KUKA KRL program: MyProgram_207().src

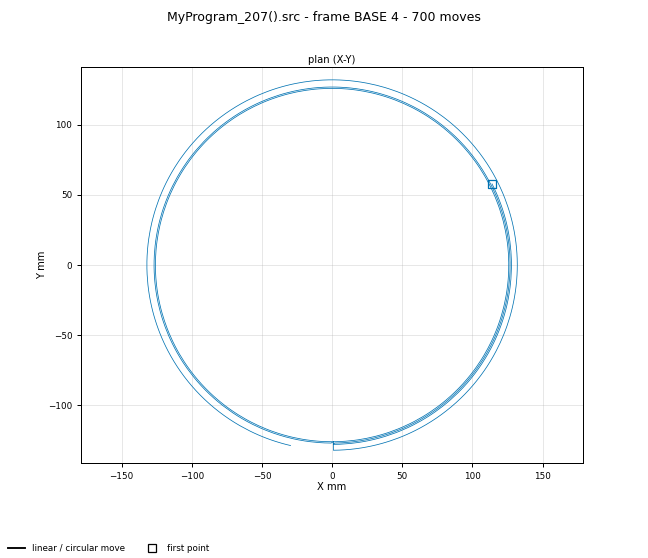
[picture p0: tool path of MyProgram_207().src in frame BASE 4, 700 of 700 moves have a stored position in this frame; points joined in program order, loops and branches not executed]
&ACCESS RVP
&REL 1
&PARAM TEMPLATE = C:\KRC\Roboter\Template\vorgabe
&PARAM EDITMASK = *
DEF MyProgram_207()
; ---- Setting reference (Base) ----
$BASE = BASE_DATA[4]

; --------------------------
; ---- Setting tool (TCP) ----
$TOOL = TOOL_DATA[3]
; --------------------------

$VEL.CP = VEL_APROX_PRINT
Startdeposition()
$VEL.CP = VEL_PRINT
LIN {X 113.9703,Y 57.8056,Z 147,A 23.526,B 22.3561,C -1.1422,E1 22.5268,E2 423.6264} C_DIS
LIN {X 115.5731,Y 54.5336,Z 147,A 21.9006,B 22.3563,C -1.138,E1 22.5287,E2 425.2529} C_DIS
LIN {X 117.0607,Y 51.2625,Z 147,A 19.7387,B 22.3577,C -1.1077,E1 22.5312,E2 427.4806} C_DIS
LIN {X 118.7833,Y 47.134,Z 147,A 18.1732,B 22.357,C -1.1224,E1 22.5328,E2 428.9979} C_DIS
LIN {X 120.2237,Y 43.3241,Z 147,A 16.48,B 22.357,C -1.1233,E1 22.5344,E2 430.6782} C_DIS
LIN {X 121.3863,Y 39.9534,Z 147,A 14.784,B 22.3574,C -1.1139,E1 22.536,E2 432.3878} C_DIS
LIN {X 122.6165,Y 35.9988,Z 147,A 13.0614,B 22.3574,C -1.1146,E1 22.5374,E2 434.0973} C_DIS
LIN {X 123.4639,Y 32.9755,Z 147,A 11.6527,B 22.3576,C -1.1103,E1 22.5384,E2 435.5083} C_DIS
LIN {X 124.3219,Y 29.5794,Z 147,A 9.9835,B 22.358,C -1.1008,E1 22.5395,E2 437.1913} C_DIS
LIN {X 125.2135,Y 25.5406,Z 147,A 8.2593,B 22.358,C -1.1012,E1 22.5405,E2 438.9031} C_DIS
LIN {X 125.8843,Y 22.0036,Z 147,A 6.6854,B 22.3582,C -1.0981,E1 22.5413,E2 440.4749} C_DIS
LIN {X 126.6501,Y 17.0512,Z 147,A 4.3479,B 22.3587,C -1.0867,E1 22.5423,E2 442.8265} C_DIS
LIN {X 127.4072,Y 9.93,Z 147,A 1.3243,B 22.3587,C -1.0853,E1 22.5431,E2 445.8334} C_DIS
LIN {X 127.7553,Y 3.0983,Z 147,A -1.7197,B 22.3592,C -1.0766,E1 22.5435,E2 448.8798} C_DIS
LIN {X 127.7807,Y -1.7513,Z 147,A -3.7775,B 22.3592,C -1.0751,E1 22.5435,E2 450.9276} C_DIS
LIN {X 127.4011,Y -10.0131,Z 147,A -7.5963,B 22.36,C -1.0579,E1 22.543,E2 454.7657} C_DIS
LIN {X 126.813,Y -15.8021,Z 147,A -10.1858,B 22.3603,C -1.0504,E1 22.5422,E2 457.3574} C_DIS
LIN {X 126.3725,Y -19.0018,Z 147,A -12.4156,B 22.3622,C -1.0089,E1 22.5412,E2 459.6807} C_DIS
LIN {X 125.461,Y -24.2979,Z 147,A -14.1841,B 22.3612,C -1.0313,E1 22.5404,E2 461.3788} C_DIS
LIN {X 124.5922,Y -28.417,Z 147,A -15.9529,B 22.3612,C -1.031,E1 22.5393,E2 463.137} C_DIS
LIN {X 123.828,Y -31.5812,Z 147,A -17.4094,B 22.3614,C -1.0265,E1 22.5383,E2 464.5956} C_DIS
LIN {X 122.7533,Y -35.5317,Z 147,A -19.2625,B 22.3617,C -1.0199,E1 22.5369,E2 466.454} C_DIS
LIN {X 121.6682,Y -39.0845,Z 147,A -20.8504,B 22.3617,C -1.0184,E1 22.5356,E2 468.0357} C_DIS
LIN {X 120.617,Y -42.2183,Z 147,A -22.4583,B 22.3622,C -1.0078,E1 22.5341,E2 469.6609} C_DIS
LIN {X 119.0143,Y -46.5442,Z 147,A -24.3866,B 22.3622,C -1.0081,E1 22.5322,E2 471.5763} C_DIS
LIN {X 117.6766,Y -49.8329,Z 147,A -25.9364,B 22.3623,C -1.0052,E1 22.5306,E2 473.124} C_DIS
LIN {X 116.3291,Y -52.904,Z 147,A -27.4435,B 22.3625,C -1.0005,E1 22.5289,E2 474.6342} C_DIS
LIN {X 115.0029,Y -55.7271,Z 147,A -29.3445,B 22.3637,C -0.9726,E1 22.5265,E2 476.5963} C_DIS
LIN {X 113.1768,Y -59.3438,Z 147,A -30.5723,B 22.3627,C -0.995,E1 22.525,E2 477.7583} C_DIS
LIN {X 111.2715,Y -62.8481,Z 147,A -32.8273,B 22.3639,C -0.9678,E1 22.5219,E2 480.071} C_DIS
LIN {X 109.42,Y -66.0186,Z 147,A -34.0958,B 22.3633,C -0.9809,E1 22.5201,E2 481.2982} C_DIS
LIN {X 106.5876,Y -70.5006,Z 147,A -36.4479,B 22.3636,C -0.9753,E1 22.5165,E2 483.6513} C_DIS
LIN {X 104.3333,Y -73.7954,Z 147,A -38.2742,B 22.3638,C -0.9687,E1 22.5136,E2 485.4848} C_DIS
LIN {X 101.8263,Y -77.2183,Z 147,A -40.7015,B 22.365,C -0.939,E1 22.5094,E2 487.9765} C_DIS
LIN {X 98.9094,Y -80.9204,Z 147,A -42.2776,B 22.3643,C -0.9585,E1 22.5068,E2 489.4933} C_DIS
LIN {X 96.1295,Y -84.2042,Z 147,A -44.5875,B 22.3652,C -0.9358,E1 22.5025,E2 491.8508} C_DIS
LIN {X 93.4028,Y -87.2188,Z 147,A -46.6124,B 22.3657,C -0.9219,E1 22.4985,E2 493.9021} C_DIS
LIN {X 89.8071,Y -90.9174,Z 147,A -48.0288,B 22.3643,C -0.958,E1 22.496,E2 495.2173} C_DIS
LIN {X 84.1748,Y -96.1551,Z 147,A -52.1641,B 22.3659,C -0.918,E1 22.4873,E2 499.4382} C_DIS
LIN {X 80.94,Y -98.8933,Z 147,A -53.3106,B 22.3646,C -0.9488,E1 22.485,E2 500.4992} C_DIS
LIN {X 78.6247,Y -100.7446,Z 147,A -54.9716,B 22.3654,C -0.9305,E1 22.4812,E2 502.2012} C_DIS
LIN {X 73.4716,Y -104.5617,Z 147,A -57.9316,B 22.3658,C -0.9207,E1 22.4745,E2 505.1751} C_DIS
LIN {X 70.6355,Y -106.4986,Z 147,A -59.2877,B 22.3655,C -0.9261,E1 22.4714,E2 506.5117} C_DIS
LIN {X 67.4689,Y -108.5317,Z 147,A -61.575,B 22.3667,C -0.8954,E1 22.4658,E2 508.8713} C_DIS
LIN {X 63.2901,Y -111.0204,Z 147,A -63.0555,B 22.3656,C -0.9236,E1 22.4625,E2 510.2728} C_DIS
LIN {X 60.2184,Y -112.7158,Z 147,A -64.7771,B 22.366,C -0.914,E1 22.4582,E2 512.0138} C_DIS
LIN {X 57.6094,Y -114.0702,Z 147,A -66.0145,B 22.366,C -0.9156,E1 22.4551,E2 513.2433} C_DIS
LIN {X 53.8834,Y -115.8764,Z 147,A -67.9484,B 22.3662,C -0.9091,E1 22.4502,E2 515.1884} C_DIS
LIN {X 47.9039,Y -118.4733,Z 147,A -70.4708,B 22.3657,C -0.9232,E1 22.4439,E2 517.667} C_DIS
LIN {X 45.3901,Y -119.4605,Z 147,A -72.0569,B 22.3664,C -0.9044,E1 22.4396,E2 519.2987} C_DIS
LIN {X 37.9509,Y -122.0278,Z 147,A -75.5995,B 22.3666,C -0.8994,E1 22.4302,E2 522.8465} C_DIS
LIN {X 34.2312,Y -123.1219,Z 147,A -77.2411,B 22.3665,C -0.9019,E1 22.4258,E2 524.4784} C_DIS
LIN {X 30.1666,Y -124.1804,Z 147,A -79.1021,B 22.3665,C -0.901,E1 22.4208,E2 526.3384} C_DIS
LIN {X 26.8694,Y -124.9351,Z 147,A -80.6062,B 22.3665,C -0.9002,E1 22.4167,E2 527.8424} C_DIS
LIN {X 23.5519,Y -125.6036,Z 147,A -82.0308,B 22.3665,C -0.9032,E1 22.4128,E2 529.2574} C_DIS
LIN {X 19.255,Y -126.3333,Z 147,A -84.2028,B 22.3669,C -0.8919,E1 22.4068,E2 531.4563} C_DIS
LIN {X 12.928,Y -127.1384,Z 147,A -86.9402,B 22.3667,C -0.8957,E1 22.3992,E2 534.1816} C_DIS
LIN {X 5.1547,Y -127.6882,Z 147,A -90.1483,B 22.3663,C -0.907,E1 22.3904,E2 537.3584} C_DIS
LIN {X 0.9063,Y -127.7615,Z 147,A -91.5691,B 22.3655,C -0.9285,E1 22.3866,E2 538.7223} C_DIS
Enddeposition()
LIN {X 0.9063,Y -127.7615,Z 147,A -91.5691,B 22.3655,C -0.9285,E1 22.3866,E2 538.7223} C_DIS
Startdeposition()
$VEL.CP = VEL_PRINT
LIN {X 1.8845,Y -126.8238,Z 147,A -90.6214,B 21.3631,C -0.7912,E1 21.3818,E2 538.0225} C_DIS
LIN {X 7.2855,Y -126.6292,Z 147,A -88.1843,B 21.3631,C -0.7918,E1 21.3886,E2 535.5846} C_DIS
LIN {X 12.6919,Y -126.2022,Z 147,A -85.9631,B 21.3634,C -0.7832,E1 21.3947,E2 533.3886} C_DIS
LIN {X 16.8635,Y -125.712,Z 147,A -83.7531,B 21.3628,C -0.7978,E1 21.4009,E2 531.1405} C_DIS
LIN {X 20.3755,Y -125.1911,Z 147,A -82.5082,B 21.3633,C -0.7834,E1 21.4042,E2 529.9366} C_DIS
LIN {X 23.4283,Y -124.6555,Z 147,A -81.3063,B 21.3636,C -0.7759,E1 21.4075,E2 528.7568} C_DIS
LIN {X 26.5889,Y -124.0192,Z 147,A -79.7344,B 21.3634,C -0.7822,E1 21.4118,E2 527.1701} C_DIS
LIN {X 29.316,Y -123.4036,Z 147,A -78.4117,B 21.3633,C -0.7859,E1 21.4154,E2 525.8395} C_DIS
LIN {X 32.5994,Y -122.5764,Z 147,A -76.8881,B 21.3633,C -0.7872,E1 21.4195,E2 524.3152} C_DIS
LIN {X 35.485,Y -121.7724,Z 147,A -75.6426,B 21.3633,C -0.7839,E1 21.4229,E2 523.081} C_DIS
LIN {X 38.1101,Y -120.9775,Z 147,A -73.9866,B 21.3626,C -0.8036,E1 21.4274,E2 521.3749} C_DIS
LIN {X 41.1624,Y -119.9729,Z 147,A -72.9028,B 21.3631,C -0.7892,E1 21.4302,E2 520.3329} C_DIS
LIN {X 44.4417,Y -118.7965,Z 147,A -71.4954,B 21.3633,C -0.784,E1 21.4338,E2 518.9434} C_DIS
LIN {X 47.2457,Y -117.7095,Z 147,A -70.1052,B 21.3633,C -0.7872,E1 21.4374,E2 517.548} C_DIS
LIN {X 50.7884,Y -116.2258,Z 147,A -67.8469,B 21.3623,C -0.8127,E1 21.4434,E2 515.2264} C_DIS
LIN {X 54.006,Y -114.7673,Z 147,A -66.4973,B 21.3626,C -0.8042,E1 21.4467,E2 513.9041} C_DIS
LIN {X 57.2234,Y -113.1956,Z 147,A -65.1958,B 21.363,C -0.7929,E1 21.4499,E2 512.6378} C_DIS
LIN {X 61.1503,Y -111.1255,Z 147,A -62.9133,B 21.3625,C -0.8085,E1 21.4556,E2 510.3204} C_DIS
LIN {X 66.7546,Y -107.852,Z 147,A -59.9734,B 21.3623,C -0.8141,E1 21.4627,E2 507.3759} C_DIS
LIN {X 70.0235,Y -105.7589,Z 147,A -58.2251,B 21.3621,C -0.8172,E1 21.4668,E2 505.626} C_DIS
LIN {X 72.9782,Y -103.7416,Z 147,A -56.6366,B 21.3621,C -0.8192,E1 21.4704,E2 504.0386} C_DIS
LIN {X 76.3709,Y -101.2699,Z 147,A -54.7572,B 21.362,C -0.8223,E1 21.4746,E2 502.1586} C_DIS
LIN {X 79.7116,Y -98.662,Z 147,A -52.906,B 21.362,C -0.8236,E1 21.4787,E2 500.3121} C_DIS
LIN {X 82.6549,Y -96.2098,Z 147,A -51.1096,B 21.3617,C -0.8303,E1 21.4825,E2 498.5056} C_DIS
LIN {X 86.242,Y -93.0081,Z 147,A -48.9386,B 21.3615,C -0.8353,E1 21.487,E2 496.3316} C_DIS
LIN {X 89.5793,Y -89.7983,Z 147,A -46.939,B 21.3615,C -0.8361,E1 21.491,E2 494.3397} C_DIS
LIN {X 93.0775,Y -86.1675,Z 147,A -44.5379,B 21.361,C -0.8472,E1 21.4956,E2 491.9207} C_DIS
LIN {X 96.2028,Y -82.6629,Z 147,A -42.5135,B 21.361,C -0.8482,E1 21.4993,E2 489.9044} C_DIS
LIN {X 98.9918,Y -79.3025,Z 147,A -40.8259,B 21.3613,C -0.8404,E1 21.5023,E2 488.2473} C_DIS
LIN {X 101.0125,Y -76.712,Z 147,A -39.0644,B 21.3607,C -0.8569,E1 21.5053,E2 486.4509} C_DIS
LIN {X 103.1861,Y -73.7614,Z 147,A -37.4465,B 21.3606,C -0.8596,E1 21.508,E2 484.8348} C_DIS
LIN {X 105.6815,Y -70.1403,Z 147,A -35.7291,B 21.3608,C -0.8529,E1 21.5106,E2 483.1459} C_DIS
LIN {X 107.4069,Y -67.4682,Z 147,A -34.0362,B 21.3602,C -0.8685,E1 21.5132,E2 481.4205} C_DIS
LIN {X 109.394,Y -64.1956,Z 147,A -32.5953,B 21.3605,C -0.8603,E1 21.5152,E2 480.0108} C_DIS
LIN {X 110.9698,Y -61.4314,Z 147,A -30.9238,B 21.36,C -0.875,E1 21.5176,E2 478.3094} C_DIS
LIN {X 113.1495,Y -57.3139,Z 147,A -28.8604,B 21.3598,C -0.8793,E1 21.5202,E2 476.2473} C_DIS
LIN {X 115.0671,Y -53.3593,Z 147,A -27.0683,B 21.3599,C -0.8764,E1 21.5224,E2 474.4747} C_DIS
LIN {X 116.2361,Y -50.7645,Z 147,A -25.578,B 21.3594,C -0.8895,E1 21.5241,E2 472.9583} C_DIS
LIN {X 117.5184,Y -47.7198,Z 147,A -24.3391,B 21.3597,C -0.8825,E1 21.5254,E2 471.7466} C_DIS
LIN {X 118.7816,Y -44.4815,Z 147,A -22.5752,B 21.3591,C -0.8961,E1 21.5271,E2 469.9573} C_DIS
LIN {X 120.1599,Y -40.6152,Z 147,A -20.6624,B 21.3588,C -0.9044,E1 21.5289,E2 468.0346} C_DIS
LIN {X 121.2727,Y -37.1565,Z 147,A -19.1074,B 21.3588,C -0.9056,E1 21.5302,E2 466.487} C_DIS
LIN {X 122.4349,Y -33.1301,Z 147,A -17.3559,B 21.3588,C -0.905,E1 21.5315,E2 464.749} C_DIS
LIN {X 123.1502,Y -30.367,Z 147,A -16.0335,B 21.3585,C -0.9105,E1 21.5324,E2 463.4205} C_DIS
LIN {X 123.8046,Y -27.5787,Z 147,A -14.5825,B 21.3581,C -0.9218,E1 21.5333,E2 461.9489} C_DIS
LIN {X 124.5256,Y -24.1076,Z 147,A -13.2442,B 21.3584,C -0.9148,E1 21.5341,E2 460.6388} C_DIS
LIN {X 125.241,Y -20.0715,Z 147,A -11.1576,B 21.3577,C -0.9314,E1 21.535,E2 458.5217} C_DIS
LIN {X 125.7775,Y -16.3637,Z 147,A -9.505,B 21.3575,C -0.935,E1 21.5357,E2 456.8709} C_DIS
LIN {X 126.3404,Y -11.2331,Z 147,A -7.2906,B 21.3575,C -0.937,E1 21.5363,E2 454.6665} C_DIS
LIN {X 126.5367,Y -8.7446,Z 147,A -5.9494,B 21.3569,C -0.9504,E1 21.5366,E2 453.2984} C_DIS
LIN {X 126.7698,Y -4.2032,Z 147,A -4.0657,B 21.3569,C -0.9491,E1 21.5368,E2 451.4315} C_DIS
LIN {X 126.8383,Y -0.4449,Z 147,A -2.4296,B 21.3569,C -0.9517,E1 21.5368,E2 449.7999} C_DIS
LIN {X 126.8228,Y 1.9441,Z 147,A -1.1678,B 21.3563,C -0.9635,E1 21.5368,E2 448.5149} C_DIS
LIN {X 126.6093,Y 7.6081,Z 147,A 1.183,B 21.3563,C -0.962,E1 21.5365,E2 446.1847} C_DIS
LIN {X 126.3642,Y 10.9505,Z 147,A 2.5647,B 21.3564,C -0.9608,E1 21.5362,E2 444.8161} C_DIS
LIN {X 125.9929,Y 14.6184,Z 147,A 4.1603,B 21.3564,C -0.9628,E1 21.5357,E2 443.2262} C_DIS
LIN {X 125.5699,Y 17.887,Z 147,A 5.8153,B 21.3558,C -0.975,E1 21.5351,E2 441.5495} C_DIS
LIN {X 124.9578,Y 21.7628,Z 147,A 7.5122,B 21.3558,C -0.9771,E1 21.5343,E2 439.8588} C_DIS
LIN {X 124.317,Y 25.1597,Z 147,A 9.1797,B 21.3553,C -0.9867,E1 21.5334,E2 438.1766} C_DIS
LIN {X 123.3874,Y 29.3829,Z 147,A 11.0808,B 21.3552,C -0.9903,E1 21.5322,E2 436.2788} C_DIS
LIN {X 122.4672,Y 33.0088,Z 147,A 12.7925,B 21.3549,C -0.9964,E1 21.531,E2 434.5622} C_DIS
LIN {X 121.3235,Y 36.9907,Z 147,A 14.5965,B 21.3548,C -0.999,E1 21.5296,E2 432.7635} C_DIS
LIN {X 120.3315,Y 40.1,Z 147,A 16.0349,B 21.3546,C -1.0018,E1 21.5283,E2 431.3273} C_DIS
LIN {X 119.4191,Y 42.7414,Z 147,A 17.5096,B 21.354,C -1.0151,E1 21.5269,E2 429.8261} C_DIS
LIN {X 117.6039,Y 47.5077,Z 147,A 19.9226,B 21.3535,C -1.0267,E1 21.5244,E2 427.3974} C_DIS
LIN {X 116.3271,Y 50.5539,Z 147,A 21.1514,B 21.3539,C -1.019,E1 21.5231,E2 426.1974} C_DIS
LIN {X 114.8228,Y 53.8878,Z 147,A 22.869,B 21.3535,C -1.0266,E1 21.5211,E2 424.4703} C_DIS
LIN {X 113.0711,Y 57.4679,Z 147,A 24.4916,B 21.3537,C -1.0236,E1 21.5191,E2 422.8661} C_DIS
LIN {X 111.6437,Y 60.1984,Z 147,A 25.8184,B 21.3537,C -1.0244,E1 21.5174,E2 421.5454} C_DIS
LIN {X 109.4873,Y 64.0369,Z 147,A 28.4643,B 21.352,C -1.0593,E1 21.5136,E2 418.8205} C_DIS
LIN {X 107.0602,Y 68.0174,Z 147,A 29.975,B 21.353,C -1.038,E1 21.5114,E2 417.3771} C_DIS
LIN {X 104.8819,Y 71.3301,Z 147,A 31.8198,B 21.3527,C -1.045,E1 21.5085,E2 415.5242} C_DIS
LIN {X 102.4325,Y 74.8053,Z 147,A 33.7868,B 21.3524,C -1.0518,E1 21.5053,E2 413.5499} C_DIS
LIN {X 99.6595,Y 78.461,Z 147,A 35.7435,B 21.3524,C -1.0516,E1 21.502,E2 411.6046} C_DIS
LIN {X 97.1625,Y 81.5326,Z 147,A 37.5801,B 21.3521,C -1.058,E1 21.4987,E2 409.7608} C_DIS
LIN {X 94.2164,Y 84.9209,Z 147,A 39.6131,B 21.3518,C -1.0628,E1 21.495,E2 407.7256} C_DIS
LIN {X 91.0186,Y 88.3389,Z 147,A 41.6737,B 21.3518,C -1.065,E1 21.491,E2 405.6694} C_DIS
LIN {X 87.95,Y 91.3951,Z 147,A 43.5616,B 21.3517,C -1.0661,E1 21.4872,E2 403.788} C_DIS
LIN {X 84.9836,Y 94.1595,Z 147,A 45.4795,B 21.3513,C -1.0736,E1 21.4833,E2 401.8588} C_DIS
LIN {X 81.8299,Y 96.9131,Z 147,A 47.3466,B 21.3512,C -1.0762,E1 21.4793,E2 399.9933} C_DIS
LIN {X 78.6628,Y 99.5009,Z 147,A 49.2351,B 21.3509,C -1.0815,E1 21.4752,E2 398.0989} C_DIS
LIN {X 75.0876,Y 102.2251,Z 147,A 51.2071,B 21.3509,C -1.0825,E1 21.4708,E2 396.1326} C_DIS
LIN {X 71.4256,Y 104.8173,Z 147,A 53.2675,B 21.3507,C -1.0874,E1 21.4661,E2 394.0672} C_DIS
LIN {X 67.7015,Y 107.2597,Z 147,A 55.0921,B 21.3509,C -1.0824,E1 21.4618,E2 392.2634} C_DIS
LIN {X 65.6014,Y 108.5568,Z 147,A 56.336,B 21.3505,C -1.0897,E1 21.4588,E2 391.0042} C_DIS
LIN {X 61.8107,Y 110.7597,Z 147,A 58.372,B 21.3503,C -1.0949,E1 21.4539,E2 388.9611} C_DIS
LIN {X 57.7877,Y 112.9083,Z 147,A 60.295,B 21.3504,C -1.0917,E1 21.4491,E2 387.0531} C_DIS
LIN {X 55.0999,Y 114.2447,Z 147,A 61.4922,B 21.3507,C -1.0866,E1 21.4462,E2 385.8739} C_DIS
LIN {X 52.5219,Y 115.4544,Z 147,A 63.0451,B 21.3501,C -1.0995,E1 21.4422,E2 384.2902} C_DIS
LIN {X 49.2412,Y 116.8893,Z 147,A 64.3472,B 21.3506,C -1.0878,E1 21.4389,E2 383.0239} C_DIS
LIN {X 46.1275,Y 118.1522,Z 147,A 65.891,B 21.3506,C -1.0905,E1 21.4349,E2 381.477} C_DIS
LIN {X 43.0582,Y 119.3049,Z 147,A 67.5406,B 21.3501,C -1.0991,E1 21.4305,E2 379.8079} C_DIS
LIN {X 39.4316,Y 120.5538,Z 147,A 69.7425,B 21.349,C -1.1206,E1 21.4246,E2 377.5521} C_DIS
LIN {X 35.589,Y 121.742,Z 147,A 71.0332,B 21.3501,C -1.0995,E1 21.4213,E2 376.3219} C_DIS
LIN {X 32.4444,Y 122.6177,Z 147,A 72.512,B 21.3501,C -1.1007,E1 21.4173,E2 374.8427} C_DIS
LIN {X 28.663,Y 123.557,Z 147,A 74.3242,B 21.3498,C -1.1039,E1 21.4123,E2 373.0248} C_DIS
LIN {X 25.4524,Y 124.2575,Z 147,A 75.8106,B 21.3498,C -1.1048,E1 21.4083,E2 371.5383} C_DIS
LIN {X 21.3949,Y 125.021,Z 147,A 77.6898,B 21.3498,C -1.1061,E1 21.4031,E2 369.6579} C_DIS
LIN {X 17.278,Y 125.6569,Z 147,A 79.6656,B 21.3495,C -1.1106,E1 21.3976,E2 367.6719} C_DIS
LIN {X 13.0799,Y 126.1622,Z 147,A 81.5158,B 21.3496,C -1.1085,E1 21.3925,E2 365.8291} C_DIS
LIN {X 9.368,Y 126.4912,Z 147,A 83.096,B 21.3498,C -1.1043,E1 21.3881,E2 364.2613} C_DIS
LIN {X 5.6663,Y 126.7127,Z 147,A 84.7258,B 21.3499,C -1.1024,E1 21.3836,E2 362.6374} C_DIS
LIN {X 2.5413,Y 126.8129,Z 147,A 86.3568,B 21.3495,C -1.1114,E1 21.379,E2 360.9821} C_DIS
LIN {X -1.518,Y 126.8299,Z 147,A 88.1668,B 21.3495,C -1.1101,E1 21.3739,E2 359.1757} C_DIS
LIN {X -5.6527,Y 126.7134,Z 147,A 90.1181,B 21.3494,C -1.113,E1 21.3685,E2 357.216} C_DIS
LIN {X -9.8605,Y 126.4552,Z 147,A 91.7492,B 21.35,C -1.101,E1 21.364,E2 355.6172} C_DIS
LIN {X -13.1058,Y 126.1594,Z 147,A 93.1324,B 21.3502,C -1.0967,E1 21.3602,E2 354.245} C_DIS
LIN {X -16.2644,Y 125.7905,Z 147,A 94.6679,B 21.35,C -1.1,E1 21.3559,E2 352.6992} C_DIS
LIN {X -20.7603,Y 125.1269,Z 147,A 96.4994,B 21.3505,C -1.0896,E1 21.3509,E2 350.8944} C_DIS
LIN {X -24.6616,Y 124.4184,Z 147,A 98.6423,B 21.3499,C -1.1026,E1 21.345,E2 348.713} C_DIS
LIN {X -27.7201,Y 123.7723,Z 147,A 100.1,B 21.3499,C -1.1033,E1 21.341,E2 347.2513} C_DIS
LIN {X -31.4319,Y 122.8812,Z 147,A 101.6902,B 21.3502,C -1.0962,E1 21.3367,E2 345.6778} C_DIS
LIN {X -35.0421,Y 121.9021,Z 147,A 103.4843,B 21.3501,C -1.0988,E1 21.3319,E2 343.8734} C_DIS
LIN {X -38.0352,Y 121.0014,Z 147,A 104.9052,B 21.3501,C -1.0976,E1 21.3281,E2 342.4528} C_DIS
LIN {X -41.575,Y 119.8298,Z 147,A 106.3171,B 21.3508,C -1.0846,E1 21.3244,E2 341.0733} C_DIS
LIN {X -44.3623,Y 118.8262,Z 147,A 107.8645,B 21.3505,C -1.0914,E1 21.3203,E2 339.5037} C_DIS
LIN {X -47.4629,Y 117.622,Z 147,A 109.3844,B 21.3505,C -1.0901,E1 21.3163,E2 337.9834} C_DIS
LIN {X -50.7011,Y 116.2635,Z 147,A 111.0935,B 21.3504,C -1.0928,E1 21.3119,E2 336.262} C_DIS
LIN {X -53.9719,Y 114.7836,Z 147,A 113.0422,B 21.3499,C -1.1035,E1 21.3069,E2 334.278} C_DIS
LIN {X -57.3652,Y 113.1234,Z 147,A 114.0368,B 21.3514,C -1.0724,E1 21.3047,E2 333.3661} C_DIS
LIN {X -61.889,Y 110.7155,Z 147,A 117.2537,B 21.3498,C -1.1046,E1 21.2965,E2 330.0496} C_DIS
LIN {X -66.0326,Y 108.2956,Z 147,A 118.9326,B 21.351,C -1.0811,E1 21.2926,E2 328.4292} C_DIS
LIN {X -69.6127,Y 106.0293,Z 147,A 120.8065,B 21.3512,C -1.076,E1 21.2883,E2 326.5623} C_DIS
LIN {X -73.3244,Y 103.4975,Z 147,A 122.7813,B 21.3515,C -1.0699,E1 21.2837,E2 324.5963} C_DIS
LIN {X -75.9784,Y 101.5652,Z 147,A 124.6517,B 21.3509,C -1.0822,E1 21.2795,E2 322.6838} C_DIS
LIN {X -78.8523,Y 99.3502,Z 147,A 125.9504,B 21.3517,C -1.0653,E1 21.2767,E2 321.4262} C_DIS
LIN {X -81.8169,Y 96.924,Z 147,A 127.5355,B 21.3522,C -1.0558,E1 21.2733,E2 319.8599} C_DIS
LIN {X -84.4057,Y 94.6778,Z 147,A 128.977,B 21.3525,C -1.0482,E1 21.2703,E2 318.4327} C_DIS
LIN {X -88.8116,Y 90.5573,Z 147,A 132.0462,B 21.3522,C -1.0554,E1 21.2641,E2 315.3286} C_DIS
LIN {X -91.657,Y 87.6762,Z 147,A 133.9648,B 21.3522,C -1.0545,E1 21.2603,E2 313.4025} C_DIS
LIN {X -97.3657,Y 81.2904,Z 147,A 137.7565,B 21.3528,C -1.0418,E1 21.2534,E2 309.6257} C_DIS
LIN {X -99.1912,Y 79.0521,Z 147,A 139.0671,B 21.353,C -1.0387,E1 21.2511,E2 308.3165} C_DIS
LIN {X -101.675,Y 75.8309,Z 147,A 140.8901,B 21.3532,C -1.0333,E1 21.248,E2 306.4979} C_DIS
LIN {X -103.4114,Y 73.4464,Z 147,A 142.3209,B 21.3532,C -1.0335,E1 21.2457,E2 305.0581} C_DIS
LIN {X -106.0078,Y 69.6454,Z 147,A 144.2176,B 21.3538,C -1.0208,E1 21.2427,E2 303.1854} C_DIS
LIN {X -108.5512,Y 65.6106,Z 147,A 146.4238,B 21.354,C -1.0168,E1 21.2395,E2 300.9768} C_DIS
LIN {X -110.3503,Y 62.5385,Z 147,A 148.1244,B 21.354,C -1.0158,E1 21.2371,E2 299.2684} C_DIS
LIN {X -112.2046,Y 59.1423,Z 147,A 149.723,B 21.3545,C -1.005,E1 21.235,E2 297.6895} C_DIS
LIN {X -113.5464,Y 56.525,Z 147,A 151.0007,B 21.3548,C -0.9992,E1 21.2334,E2 296.4197} C_DIS
LIN {X -115.2278,Y 53.0118,Z 147,A 153.0207,B 21.3545,C -1.0041,E1 21.231,E2 294.373} C_DIS
LIN {X -117.0658,Y 48.8187,Z 147,A 154.9862,B 21.355,C -0.9939,E1 21.2288,E2 292.4226} C_DIS
LIN {X -118.5773,Y 45.0267,Z 147,A 157.1165,B 21.3548,C -0.9994,E1 21.2267,E2 290.2629} C_DIS
LIN {X -120.1187,Y 40.739,Z 147,A 159.0352,B 21.3553,C -0.9877,E1 21.2249,E2 288.3636} C_DIS
LIN {X -121.198,Y 37.4006,Z 147,A 160.5298,B 21.3556,C -0.9794,E1 21.2237,E2 286.8818} C_DIS
LIN {X -122.871,Y 31.4722,Z 147,A 163.3581,B 21.3559,C -0.9725,E1 21.2216,E2 284.0529} C_DIS
LIN {X -123.6444,Y 28.2802,Z 147,A 164.7918,B 21.3562,C -0.9659,E1 21.2207,E2 282.6274} C_DIS
LIN {X -124.325,Y 25.1205,Z 147,A 166.4099,B 21.3562,C -0.9674,E1 21.2197,E2 280.9938} C_DIS
LIN {X -125.118,Y 20.8135,Z 147,A 168.3115,B 21.3566,C -0.9582,E1 21.2188,E2 279.1042} C_DIS
LIN {X -125.6629,Y 17.236,Z 147,A 170.0014,B 21.3566,C -0.9551,E1 21.2181,E2 277.4107} C_DIS
LIN {X -126.1089,Y 13.5752,Z 147,A 171.648,B 21.3569,C -0.9491,E1 21.2176,E2 275.769} C_DIS
LIN {X -126.4759,Y 9.5777,Z 147,A 173.3626,B 21.3573,C -0.9396,E1 21.2172,E2 274.0685} C_DIS
LIN {X -126.6451,Y 7.0145,Z 147,A 174.7931,B 21.3571,C -0.9463,E1 21.217,E2 272.6092} C_DIS
LIN {X -126.804,Y 2.9711,Z 147,A 176.5928,B 21.3573,C -0.9394,E1 21.2168,E2 270.8156} C_DIS
LIN {X -126.8311,Y -1.4468,Z 147,A 178.5295,B 21.3577,C -0.9308,E1 21.2168,E2 268.8889} C_DIS
LIN {X -126.7387,Y -5.0089,Z 147,A -179.8791,B 21.3579,C -0.925,E1 21.217,E2 267.3021} C_DIS
LIN {X -126.5168,Y -9.0168,Z 147,A -178.1018,B 21.3582,C -0.9179,E1 21.2173,E2 265.5316} C_DIS
LIN {X -126.2436,Y -12.2609,Z 147,A -176.5153,B 21.3582,C -0.9177,E1 21.2177,E2 263.9342} C_DIS
LIN {X -125.7846,Y -16.3094,Z 147,A -174.8337,B 21.3587,C -0.9058,E1 21.2183,E2 262.2735} C_DIS
LIN {X -125.3527,Y -19.3504,Z 147,A -173.4235,B 21.3589,C -0.9024,E1 21.2188,E2 260.8628} C_DIS
LIN {X -124.7951,Y -22.6715,Z 147,A -171.664,B 21.3587,C -0.9069,E1 21.2197,E2 259.0783} C_DIS
LIN {X -124.0023,Y -26.6673,Z 147,A -169.9438,B 21.3591,C -0.8966,E1 21.2207,E2 257.3745} C_DIS
LIN {X -123.2772,Y -29.8405,Z 147,A -168.4322,B 21.3592,C -0.8937,E1 21.2216,E2 255.8603} C_DIS
LIN {X -122.6152,Y -32.4538,Z 147,A -166.695,B 21.3585,C -0.9103,E1 21.2229,E2 254.0652} C_DIS
LIN {X -121.4257,Y -36.6565,Z 147,A -165.226,B 21.3596,C -0.8847,E1 21.2241,E2 252.6569} C_DIS
LIN {X -120.4041,Y -39.8818,Z 147,A -163.1202,B 21.3589,C -0.9028,E1 21.226,E2 250.4868} C_DIS
LIN {X -118.8884,Y -44.1962,Z 147,A -161.801,B 21.3602,C -0.8675,E1 21.2271,E2 249.256} C_DIS
LIN {X -117.6839,Y -47.3093,Z 147,A -160.119,B 21.3602,C -0.87,E1 21.2289,E2 247.5562} C_DIS
LIN {X -116.5005,Y -50.1529,Z 147,A -158.8173,B 21.3604,C -0.8625,E1 21.2303,E2 246.2665} C_DIS
LIN {X -115.456,Y -52.5184,Z 147,A -157.552,B 21.3604,C -0.863,E1 21.2317,E2 244.9916} C_DIS
LIN {X -113.8661,Y -55.8768,Z 147,A -155.829,B 21.3605,C -0.8601,E1 21.2338,E2 243.2654} C_DIS
LIN {X -112.0256,Y -59.483,Z 147,A -154.1184,B 21.3609,C -0.8504,E1 21.236,E2 241.5706} C_DIS
LIN {X -110.4503,Y -62.3612,Z 147,A -152.421,B 21.3607,C -0.8549,E1 21.2383,E2 239.8502} C_DIS
LIN {X -108.3915,Y -65.8748,Z 147,A -150.5605,B 21.3609,C -0.8509,E1 21.241,E2 237.9893} C_DIS
LIN {X -106.3198,Y -69.1682,Z 147,A -148.808,B 21.3611,C -0.8462,E1 21.2436,E2 236.2393} C_DIS
LIN {X -103.3268,Y -73.5647,Z 147,A -146.7004,B 21.3617,C -0.8285,E1 21.2469,E2 234.168} C_DIS
LIN {X -98.6568,Y -79.718,Z 147,A -142.9187,B 21.3617,C -0.8316,E1 21.2534,E2 230.3564} C_DIS
LIN {X -96.1393,Y -82.7366,Z 147,A -141.1053,B 21.3617,C -0.829,E1 21.2567,E2 228.5403} C_DIS
LIN {X -93.3895,Y -85.8285,Z 147,A -139.2387,B 21.3619,C -0.8247,E1 21.2602,E2 226.6756} C_DIS
LIN {X -90.5284,Y -88.841,Z 147,A -137.3227,B 21.3619,C -0.8223,E1 21.2639,E2 224.7565} C_DIS
LIN {X -87.5968,Y -91.7329,Z 147,A -135.5026,B 21.3622,C -0.8168,E1 21.2675,E2 222.9424} C_DIS
LIN {X -84.5646,Y -94.5355,Z 147,A -133.6279,B 21.3622,C -0.8135,E1 21.2714,E2 221.068} C_DIS
LIN {X -81.5422,Y -97.1545,Z 147,A -131.7656,B 21.3623,C -0.8123,E1 21.2754,E2 219.2003} C_DIS
LIN {X -77.7964,Y -100.1791,Z 147,A -129.6511,B 21.3625,C -0.8059,E1 21.28,E2 217.0942} C_DIS
LIN {X -70.7902,Y -105.2474,Z 147,A -125.629,B 21.3626,C -0.8039,E1 21.2892,E2 213.0608} C_DIS
LIN {X -67.2463,Y -107.546,Z 147,A -123.7526,B 21.3628,C -0.7997,E1 21.2935,E2 211.189} C_DIS
LIN {X -63.998,Y -109.5101,Z 147,A -121.9923,B 21.3628,C -0.7991,E1 21.2978,E2 209.4241} C_DIS
LIN {X -60.2719,Y -111.6042,Z 147,A -120.0126,B 21.3628,C -0.7985,E1 21.3026,E2 207.4392} C_DIS
LIN {X -56.4597,Y -113.5785,Z 147,A -118.1934,B 21.3631,C -0.7911,E1 21.3071,E2 205.6345} C_DIS
LIN {X -53.2215,Y -115.1308,Z 147,A -116.6636,B 21.3633,C -0.7854,E1 21.311,E2 204.1158} C_DIS
LIN {X -50.917,Y -116.1702,Z 147,A -115.3238,B 21.363,C -0.7923,E1 21.3145,E2 202.7533} C_DIS
LIN {X -47.842,Y -117.4692,Z 147,A -114.0927,B 21.3635,C -0.7793,E1 21.3175,E2 201.5545} C_DIS
LIN {X -44.7059,Y -118.6975,Z 147,A -112.4736,B 21.3634,C -0.7819,E1 21.3218,E2 199.9242} C_DIS
LIN {X -41.9917,Y -119.685,Z 147,A -110.4104,B 21.3623,C -0.8124,E1 21.3275,E2 197.7725} C_DIS
LIN {X -37.1664,Y -121.2697,Z 147,A -108.7393,B 21.3633,C -0.7846,E1 21.3317,E2 196.1743} C_DIS
LIN {X -33.1194,Y -122.4377,Z 147,A -106.8796,B 21.3634,C -0.7815,E1 21.3367,E2 194.3196} C_DIS
LIN {X -29.9233,Y -123.2572,Z 147,A -105.5295,B 21.3636,C -0.7748,E1 21.3403,E2 192.9857} C_DIS
LIN {X -27.4827,Y -123.8263,Z 147,A -104.1529,B 21.3633,C -0.7844,E1 21.3442,E2 191.5805} C_DIS
LIN {X -23.8146,Y -124.5816,Z 147,A -102.6949,B 21.3637,C -0.7739,E1 21.3481,E2 190.1494} C_DIS
LIN {X -19.4147,Y -125.3427,Z 147,A -100.6287,B 21.3637,C -0.7753,E1 21.3538,E2 188.077} C_DIS
LIN {X -15.7251,Y -125.8609,Z 147,A -98.8317,B 21.3635,C -0.7797,E1 21.3588,E2 186.2664} C_DIS
LIN {X -12.1995,Y -126.2495,Z 147,A -97.411,B 21.3637,C -0.7719,E1 21.3627,E2 184.8662} C_DIS
LIN {X -9.3769,Y -126.4905,Z 147,A -95.9925,B 21.3635,C -0.7777,E1 21.3667,E2 183.4311} C_DIS
LIN {X -5.2978,Y -126.7274,Z 147,A -93.9712,B 21.3633,C -0.7852,E1 21.3724,E2 181.3885} C_DIS
LIN {X -0.7396,Y -126.8355,Z 147,A -92.1036,B 21.3636,C -0.7774,E1 21.3775,E2 179.5423} C_DIS
LIN {X -0.7396,Y -126.8355,Z 147,A -92.1036,B 21.3636,C -0.7774,E1 21.3775,E2 179.5423} C_DIS
Enddeposition()
LIN {X 0.8881,Y -125.8783,Z 147,A -91.3008,B 20.2634,C -0.6186,E1 20.2743,E2 179.0628} C_DIS
Startdeposition()
$VEL.CP = VEL_PRINT
LIN {X -1.28,Y -125.878,Z 147,A -92.7137,B 20.2639,C -0.6014,E1 20.2702,E2 180.5251} C_DIS
LIN {X -4.3969,Y -125.8073,Z 147,A -94.1696,B 20.2639,C -0.5999,E1 20.2661,E2 181.9857} C_DIS
LIN {X -7.4722,Y -125.6614,Z 147,A -95.5006,B 20.2639,C -0.6026,E1 20.2624,E2 183.3093} C_DIS
LIN {X -10.8085,Y -125.4183,Z 147,A -96.9698,B 20.2639,C -0.6048,E1 20.2583,E2 184.773} C_DIS
LIN {X -14.1427,Y -125.0878,Z 147,A -98.7047,B 20.2641,C -0.5968,E1 20.2535,E2 186.5324} C_DIS
LIN {X -18.211,Y -124.5594,Z 147,A -100.4253,B 20.2639,C -0.6029,E1 20.2487,E2 188.2368} C_DIS
LIN {X -21.5202,Y -124.0315,Z 147,A -101.8946,B 20.2639,C -0.6056,E1 20.2447,E2 189.7002} C_DIS
LIN {X -24.562,Y -123.4646,Z 147,A -103.2565,B 20.2637,C -0.608,E1 20.241,E2 191.057} C_DIS
LIN {X -27.3195,Y -122.8848,Z 147,A -104.6384,B 20.2638,C -0.6047,E1 20.2372,E2 192.4505} C_DIS
LIN {X -30.2825,Y -122.1882,Z 147,A -106.1257,B 20.2639,C -0.6015,E1 20.2331,E2 193.9495} C_DIS
LIN {X -34.3003,Y -121.1203,Z 147,A -108.0068,B 20.2639,C -0.6032,E1 20.2281,E2 195.8295} C_DIS
LIN {X -38.0606,Y -119.9913,Z 147,A -109.7407,B 20.2638,C -0.6066,E1 20.2234,E2 197.5574} C_DIS
LIN {X -41.0397,Y -119.0052,Z 147,A -111.0414,B 20.2636,C -0.6126,E1 20.22,E2 198.8436} C_DIS
LIN {X -43.2096,Y -118.2357,Z 147,A -112.2507,B 20.2638,C -0.6074,E1 20.2168,E2 200.0711} C_DIS
LIN {X -46.5023,Y -116.9801,Z 147,A -113.8752,B 20.2638,C -0.6081,E1 20.2126,E2 201.6979} C_DIS
LIN {X -49.5968,Y -115.7011,Z 147,A -115.3192,B 20.2636,C -0.6128,E1 20.2089,E2 203.1325} C_DIS
LIN {X -52.4241,Y -114.448,Z 147,A -116.7302,B 20.2636,C -0.6142,E1 20.2053,E2 204.5437} C_DIS
LIN {X -55.2142,Y -113.1287,Z 147,A -118.1364,B 20.2636,C -0.6158,E1 20.2018,E2 205.9498} C_DIS
LIN {X -57.9708,Y -111.7416,Z 147,A -119.5952,B 20.2636,C -0.6155,E1 20.1981,E2 207.4145} C_DIS
LIN {X -61.3921,Y -109.9,Z 147,A -121.4391,B 20.2636,C -0.615,E1 20.1936,E2 209.2663} C_DIS
LIN {X -64.4924,Y -108.1093,Z 147,A -122.9626,B 20.2633,C -0.6214,E1 20.1899,E2 210.7774} C_DIS
LIN {X -66.7419,Y -106.7356,Z 147,A -124.2652,B 20.2634,C -0.6193,E1 20.1868,E2 212.0911} C_DIS
LIN {X -69.4718,Y -104.9793,Z 147,A -125.797,B 20.2634,C -0.6196,E1 20.1832,E2 213.6285} C_DIS
LIN {X -72.548,Y -102.877,Z 147,A -127.276,B 20.2631,C -0.6304,E1 20.1799,E2 215.0822} C_DIS
LIN {X -75.0134,Y -101.0937,Z 147,A -128.685,B 20.2631,C -0.6319,E1 20.1767,E2 216.4932} C_DIS
LIN {X -77.7173,Y -99.0299,Z 147,A -130.4054,B 20.2631,C -0.6282,E1 20.1729,E2 218.2322} C_DIS
LIN {X -81.0521,Y -96.3197,Z 147,A -132.3992,B 20.2631,C -0.6304,E1 20.1686,E2 220.2291} C_DIS
LIN {X -84.0125,Y -93.7486,Z 147,A -134.203,B 20.263,C -0.6332,E1 20.1648,E2 222.0339} C_DIS
LIN {X -86.8971,Y -91.0813,Z 147,A -135.979,B 20.2629,C -0.6373,E1 20.1612,E2 223.8074} C_DIS
LIN {X -90.1004,Y -87.9143,Z 147,A -138.0829,B 20.2629,C -0.6396,E1 20.157,E2 225.9158} C_DIS
LIN {X -93.1803,Y -84.6424,Z 147,A -140.0058,B 20.2625,C -0.6485,E1 20.1534,E2 227.8234} C_DIS
LIN {X -95.737,Y -81.7398,Z 147,A -141.8745,B 20.2625,C -0.6485,E1 20.15,E2 229.7029} C_DIS
LIN {X -98.3357,Y -78.5942,Z 147,A -143.7581,B 20.2625,C -0.6519,E1 20.1467,E2 231.5878} C_DIS
LIN {X -101.1254,Y -74.9708,Z 147,A -145.7534,B 20.2622,C -0.66,E1 20.1433,E2 233.5716} C_DIS
LIN {X -103.3231,Y -71.9113,Z 147,A -147.5457,B 20.2622,C -0.6614,E1 20.1404,E2 235.3709} C_DIS
LIN {X -105.3749,Y -68.8707,Z 147,A -149.1835,B 20.262,C -0.6667,E1 20.1379,E2 237.0036} C_DIS
LIN {X -107.1725,Y -66.0381,Z 147,A -150.5919,B 20.2617,C -0.6749,E1 20.1358,E2 238.3971} C_DIS
LIN {X -108.759,Y -63.3917,Z 147,A -152.0553,B 20.2617,C -0.6765,E1 20.1337,E2 239.8656} C_DIS
LIN {X -110.1535,Y -60.9353,Z 147,A -153.3606,B 20.2616,C -0.6792,E1 20.1319,E2 241.1718} C_DIS
LIN {X -111.7358,Y -57.9819,Z 147,A -154.8871,B 20.2614,C -0.6832,E1 20.13,E2 242.6967} C_DIS
LIN {X -113.6835,Y -54.0604,Z 147,A -156.9061,B 20.2613,C -0.6878,E1 20.1275,E2 244.7163} C_DIS
LIN {X -114.9752,Y -51.2557,Z 147,A -158.3205,B 20.2612,C -0.6914,E1 20.1258,E2 246.13} C_DIS
LIN {X -116.197,Y -48.422,Z 147,A -159.7261,B 20.261,C -0.6953,E1 20.1243,E2 247.5341} C_DIS
LIN {X -117.4488,Y -45.3026,Z 147,A -161.2768,B 20.261,C -0.6989,E1 20.1227,E2 249.0852} C_DIS
LIN {X -118.5316,Y -42.3888,Z 147,A -162.7011,B 20.2608,C -0.7026,E1 20.1214,E2 250.5088} C_DIS
LIN {X -119.4478,Y -39.7325,Z 147,A -163.9886,B 20.2607,C -0.7061,E1 20.1202,E2 251.7956} C_DIS
LIN {X -120.4609,Y -36.5475,Z 147,A -165.5212,B 20.2606,C -0.7101,E1 20.1189,E2 253.3275} C_DIS
LIN {X -121.2452,Y -33.8538,Z 147,A -166.7342,B 20.2603,C -0.7162,E1 20.118,E2 254.5317} C_DIS
LIN {X -122.0449,Y -30.8467,Z 147,A -168.2735,B 20.2603,C -0.7161,E1 20.1169,E2 256.0828} C_DIS
LIN {X -122.8835,Y -27.325,Z 147,A -170.0596,B 20.2603,C -0.7161,E1 20.1158,E2 257.8821} C_DIS
LIN {X -123.7081,Y -23.3007,Z 147,A -171.8003,B 20.26,C -0.7264,E1 20.1149,E2 259.6058} C_DIS
LIN {X -124.2421,Y -20.2639,Z 147,A -173.1881,B 20.2598,C -0.7312,E1 20.1142,E2 260.9899} C_DIS
LIN {X -124.7386,Y -16.9452,Z 147,A -174.8361,B 20.2598,C -0.7316,E1 20.1136,E2 262.6492} C_DIS
LIN {X -125.1747,Y -13.3353,Z 147,A -176.5352,B 20.2597,C -0.7352,E1 20.113,E2 264.3507} C_DIS
LIN {X -125.5616,Y -8.9912,Z 147,A -178.5536,B 20.2595,C -0.7402,E1 20.1126,E2 266.3699} C_DIS
LIN {X -125.7875,Y -4.9051,Z 147,A 179.6787,B 20.2592,C -0.7494,E1 20.1123,E2 268.1243} C_DIS
LIN {X -125.8702,Y -1.8232,Z 147,A 178.3437,B 20.259,C -0.7562,E1 20.1123,E2 269.4497} C_DIS
LIN {X -125.8748,Y 1.5468,Z 147,A 176.8327,B 20.2588,C -0.7619,E1 20.1123,E2 270.9558} C_DIS
LIN {X -125.8085,Y 4.3661,Z 147,A 175.3727,B 20.2588,C -0.7596,E1 20.1124,E2 272.4335} C_DIS
LIN {X -125.6629,Y 7.4479,Z 147,A 174.0356,B 20.2586,C -0.7664,E1 20.1126,E2 273.7609} C_DIS
LIN {X -125.4389,Y 10.5649,Z 147,A 172.6159,B 20.2584,C -0.771,E1 20.1129,E2 275.1781} C_DIS
LIN {X -125.1456,Y 13.6057,Z 147,A 171.1935,B 20.2584,C -0.7742,E1 20.1133,E2 276.6019} C_DIS
LIN {X -124.739,Y 16.9428,Z 147,A 169.689,B 20.2581,C -0.7799,E1 20.1138,E2 278.1012} C_DIS
LIN {X -124.2869,Y 19.9952,Z 147,A 168.2374,B 20.258,C -0.7826,E1 20.1145,E2 279.5558} C_DIS
LIN {X -123.8077,Y 22.7712,Z 147,A 166.8941,B 20.258,C -0.7845,E1 20.1151,E2 280.9039} C_DIS
LIN {X -123.2132,Y 25.7973,Z 147,A 165.5451,B 20.2577,C -0.7908,E1 20.1159,E2 282.2446} C_DIS
LIN {X -122.6059,Y 28.5403,Z 147,A 164.2072,B 20.2577,C -0.7926,E1 20.1167,E2 283.587} C_DIS
LIN {X -121.7201,Y 32.1061,Z 147,A 162.5649,B 20.2574,C -0.7989,E1 20.1178,E2 285.2233} C_DIS
LIN {X -120.8983,Y 35.0736,Z 147,A 161.244,B 20.2571,C -0.806,E1 20.1188,E2 286.5331} C_DIS
LIN {X -120.0844,Y 37.7691,Z 147,A 159.7808,B 20.2572,C -0.8035,E1 20.12,E2 288.0144} C_DIS
LIN {X -119.037,Y 40.948,Z 147,A 158.422,B 20.2568,C -0.8139,E1 20.1212,E2 289.3525} C_DIS
LIN {X -118.0945,Y 43.5947,Z 147,A 157.0305,B 20.2568,C -0.8138,E1 20.1226,E2 290.7545} C_DIS
LIN {X -116.9825,Y 46.4964,Z 147,A 155.4644,B 20.2568,C -0.8126,E1 20.1242,E2 292.3351} C_DIS
LIN {X -115.3677,Y 50.3678,Z 147,A 153.5418,B 20.2567,C -0.8178,E1 20.1263,E2 294.2561} C_DIS
LIN {X -113.7902,Y 53.8371,Z 147,A 151.9456,B 20.2563,C -0.8277,E1 20.1281,E2 295.8344} C_DIS
LIN {X -112.6767,Y 56.1304,Z 147,A 150.6742,B 20.2563,C -0.8271,E1 20.1297,E2 297.1161} C_DIS
LIN {X -111.1446,Y 59.1077,Z 147,A 149.2343,B 20.256,C -0.8344,E1 20.1316,E2 298.5445} C_DIS
LIN {X -109.5341,Y 62.0429,Z 147,A 147.7336,B 20.2558,C -0.8396,E1 20.1336,E2 300.0402} C_DIS
LIN {X -108.1207,Y 64.4734,Z 147,A 146.4119,B 20.2558,C -0.8416,E1 20.1355,E2 301.3646} C_DIS
LIN {X -106.5121,Y 67.0976,Z 147,A 145.0855,B 20.2555,C -0.8482,E1 20.1374,E2 302.6805} C_DIS
LIN {X -104.7532,Y 69.8117,Z 147,A 143.4842,B 20.2555,C -0.8475,E1 20.1399,E2 304.2939} C_DIS
LIN {X -102.915,Y 72.4943,Z 147,A 142.1057,B 20.2552,C -0.8551,E1 20.1421,E2 305.659} C_DIS
LIN {X -101.11,Y 74.9915,Z 147,A 140.6215,B 20.2552,C -0.8558,E1 20.1445,E2 307.1501} C_DIS
LIN {X -98.8643,Y 77.9281,Z 147,A 138.8696,B 20.2551,C -0.8577,E1 20.1475,E2 308.907} C_DIS
LIN {X -96.2937,Y 81.0831,Z 147,A 136.9239,B 20.2551,C -0.859,E1 20.151,E2 310.8603} C_DIS
LIN {X -93.7825,Y 83.9746,Z 147,A 135.148,B 20.2549,C -0.8621,E1 20.1543,E2 312.6373} C_DIS
LIN {X -90.6345,Y 87.3634,Z 147,A 133.1529,B 20.2545,C -0.8711,E1 20.1581,E2 314.6172} C_DIS
LIN {X -87.8592,Y 90.1544,Z 147,A 131.2203,B 20.2545,C -0.8701,E1 20.1619,E2 316.5629} C_DIS
LIN {X -84.6271,Y 93.1941,Z 147,A 129.3252,B 20.2542,C -0.8792,E1 20.1658,E2 318.4415} C_DIS
LIN {X -81.7357,Y 95.7405,Z 147,A 127.4347,B 20.2542,C -0.878,E1 20.1698,E2 320.3446} C_DIS
LIN {X -78.6613,Y 98.2824,Z 147,A 125.599,B 20.2542,C -0.8811,E1 20.1738,E2 322.1802} C_DIS
LIN {X -75.0874,Y 101.0386,Z 147,A 123.7242,B 20.2537,C -0.8918,E1 20.1779,E2 324.0325} C_DIS
LIN {X -72.4906,Y 102.9176,Z 147,A 122.296,B 20.2535,C -0.8958,E1 20.1811,E2 325.4554} C_DIS
LIN {X -70.1587,Y 104.5216,Z 147,A 120.7771,B 20.2538,C -0.8898,E1 20.1847,E2 326.9982} C_DIS
LIN {X -66.3369,Y 106.9876,Z 147,A 118.758,B 20.2535,C -0.8954,E1 20.1894,E2 329.0091} C_DIS
LIN {X -63.3176,Y 108.802,Z 147,A 117.2554,B 20.2532,C -0.9018,E1 20.193,E2 330.4987} C_DIS
LIN {X -60.8942,Y 110.1763,Z 147,A 115.9728,B 20.2532,C -0.9034,E1 20.1961,E2 331.7815} C_DIS
LIN {X -57.9697,Y 111.7422,Z 147,A 114.4626,B 20.2531,C -0.9058,E1 20.1999,E2 333.2899} C_DIS
LIN {X -55.4717,Y 113.0016,Z 147,A 113.1688,B 20.2531,C -0.907,E1 20.2031,E2 334.5845} C_DIS
LIN {X -52.6562,Y 114.3407,Z 147,A 111.75,B 20.2529,C -0.9091,E1 20.2067,E2 336.0018} C_DIS
LIN {X -49.8386,Y 115.5965,Z 147,A 110.3416,B 20.2529,C -0.9109,E1 20.2103,E2 337.4092} C_DIS
LIN {X -46.9909,Y 116.7831,Z 147,A 108.8896,B 20.2529,C -0.911,E1 20.214,E2 338.865} C_DIS
LIN {X -43.8636,Y 117.9937,Z 147,A 107.4011,B 20.2527,C -0.9143,E1 20.2179,E2 340.3479} C_DIS
LIN {X -40.9584,Y 119.0334,Z 147,A 106.035,B 20.2526,C -0.9174,E1 20.2215,E2 341.7083} C_DIS
LIN {X -38.2862,Y 119.9192,Z 147,A 104.6114,B 20.2527,C -0.9135,E1 20.2253,E2 343.1465} C_DIS
LIN {X -33.8248,Y 121.2533,Z 147,A 102.5831,B 20.2525,C -0.9191,E1 20.2307,E2 345.1628} C_DIS
LIN {X -30.8407,Y 122.0465,Z 147,A 101.138,B 20.2525,C -0.9189,E1 20.2346,E2 346.6111} C_DIS
LIN {X -27.5808,Y 122.8251,Z 147,A 99.6506,B 20.2524,C -0.9216,E1 20.2387,E2 348.0931} C_DIS
LIN {X -25.1985,Y 123.3351,Z 147,A 98.4631,B 20.2524,C -0.9196,E1 20.2419,E2 349.2884} C_DIS
LIN {X -21.5048,Y 124.0343,Z 147,A 96.8368,B 20.2523,C -0.9239,E1 20.2464,E2 350.9041} C_DIS
LIN {X -18.8859,Y 124.4587,Z 147,A 95.5435,B 20.2523,C -0.9215,E1 20.25,E2 352.2059} C_DIS
LIN {X -15.6715,Y 124.9056,Z 147,A 94.1291,B 20.2523,C -0.9247,E1 20.2539,E2 353.6124} C_DIS
LIN {X -12.6349,Y 125.2488,Z 147,A 92.639,B 20.2523,C -0.9216,E1 20.258,E2 355.1126} C_DIS
LIN {X -9.523,Y 125.5228,Z 147,A 91.2461,B 20.2523,C -0.9232,E1 20.2619,E2 356.5014} C_DIS
LIN {X -6.1669,Y 125.732,Z 147,A 89.8343,B 20.2521,C -0.9283,E1 20.2658,E2 357.8992} C_DIS
LIN {X -3.0848,Y 125.846,Z 147,A 88.4193,B 20.2521,C -0.9282,E1 20.2697,E2 359.3147} C_DIS
LIN {X -0.0018,Y 125.8851,Z 147,A 87.0048,B 20.2521,C -0.928,E1 20.2737,E2 360.7297} C_DIS
LIN {X 3.1041,Y 125.8454,Z 147,A 85.632,B 20.2521,C -0.9297,E1 20.2775,E2 362.0974} C_DIS
LIN {X 6.1862,Y 125.7311,Z 147,A 84.0521,B 20.2523,C -0.9229,E1 20.282,E2 363.6962} C_DIS
LIN {X 10.75,Y 125.4233,Z 147,A 82.1147,B 20.2521,C -0.9284,E1 20.2873,E2 365.6168} C_DIS
LIN {X 13.5956,Y 125.1467,Z 147,A 80.7412,B 20.2522,C -0.9253,E1 20.2912,E2 366.9978} C_DIS
LIN {X 16.9431,Y 124.7389,Z 147,A 79.2636,B 20.2522,C -0.9272,E1 20.2952,E2 368.4686} C_DIS
LIN {X 20.0036,Y 124.2855,Z 147,A 77.8208,B 20.2522,C -0.9253,E1 20.2992,E2 369.915} C_DIS
LIN {X 22.7803,Y 123.806,Z 147,A 76.4887,B 20.2523,C -0.9229,E1 20.3029,E2 371.2523} C_DIS
LIN {X 25.8047,Y 123.2117,Z 147,A 75.1532,B 20.2523,C -0.9248,E1 20.3065,E2 372.58} C_DIS
LIN {X 28.8338,Y 122.538,Z 147,A 73.7354,B 20.2523,C -0.9238,E1 20.3104,E2 373.9983} C_DIS
LIN {X 31.3262,Y 121.9233,Z 147,A 72.4102,B 20.2526,C -0.917,E1 20.314,E2 375.3407} C_DIS
LIN {X 35.061,Y 120.902,Z 147,A 70.8968,B 20.2522,C -0.9255,E1 20.318,E2 376.8262} C_DIS
LIN {X 37.9674,Y 120.0211,Z 147,A 69.2525,B 20.2527,C -0.9141,E1 20.3225,E2 378.4998} C_DIS
LIN {X 42.0784,Y 118.6435,Z 147,A 67.4334,B 20.2525,C -0.9184,E1 20.3272,E2 380.3018} C_DIS
LIN {X 45.0595,Y 117.5433,Z 147,A 66.0267,B 20.2525,C -0.9186,E1 20.3309,E2 381.7042} C_DIS
LIN {X 48.1776,Y 116.2991,Z 147,A 64.5014,B 20.2525,C -0.9172,E1 20.3349,E2 383.2293} C_DIS
LIN {X 51.0143,Y 115.0832,Z 147,A 63.1025,B 20.2526,C -0.9158,E1 20.3384,E2 384.6278} C_DIS
LIN {X 53.8203,Y 113.7982,Z 147,A 61.7032,B 20.2527,C -0.9144,E1 20.342,E2 386.0267} C_DIS
LIN {X 56.5936,Y 112.4452,Z 147,A 60.3056,B 20.2527,C -0.9129,E1 20.3455,E2 387.4239} C_DIS
LIN {X 58.8884,Y 111.2598,Z 147,A 59.0636,B 20.253,C -0.9087,E1 20.3486,E2 388.6736} C_DIS
LIN {X 62.0539,Y 109.5279,Z 147,A 57.3531,B 20.2532,C -0.9036,E1 20.3528,E2 390.3924} C_DIS
LIN {X 65.8107,Y 107.3119,Z 147,A 55.5488,B 20.253,C -0.908,E1 20.357,E2 392.177} C_DIS
LIN {X 68.4227,Y 105.6658,Z 147,A 54.0561,B 20.2532,C -0.9022,E1 20.3606,E2 393.6801} C_DIS
LIN {X 71.213,Y 103.8056,Z 147,A 52.5946,B 20.2532,C -0.9024,E1 20.3639,E2 395.1351} C_DIS
LIN {X 73.5171,Y 102.1874,Z 147,A 51.3878,B 20.2532,C -0.9032,E1 20.3667,E2 396.3341} C_DIS
LIN {X 76.2329,Y 100.1776,Z 147,A 49.6343,B 20.2537,C -0.8917,E1 20.3706,E2 398.1126} C_DIS
LIN {X 79.37,Y 97.711,Z 147,A 47.8179,B 20.2538,C -0.8884,E1 20.3746,E2 399.93} C_DIS
LIN {X 82.7056,Y 94.9035,Z 147,A 45.8499,B 20.2539,C -0.8852,E1 20.3788,E2 401.8974} C_DIS
LIN {X 85.6831,Y 92.2243,Z 147,A 44.0383,B 20.2541,C -0.882,E1 20.3825,E2 403.7088} C_DIS
LIN {X 88.6198,Y 89.4061,Z 147,A 42.4084,B 20.2539,C -0.8873,E1 20.3857,E2 405.315} C_DIS
LIN {X 91.0741,Y 86.9047,Z 147,A 40.6729,B 20.2542,C -0.8781,E1 20.3891,E2 407.0676} C_DIS
LIN {X 93.8817,Y 83.8639,Z 147,A 38.757,B 20.2545,C -0.8726,E1 20.3927,E2 408.9885} C_DIS
LIN {X 96.7303,Y 80.5622,Z 147,A 36.8839,B 20.2545,C -0.8726,E1 20.3961,E2 410.8508} C_DIS
LIN {X 99.1525,Y 77.5612,Z 147,A 35.1216,B 20.2547,C -0.8682,E1 20.3992,E2 412.6154} C_DIS
LIN {X 101.6576,Y 74.2479,Z 147,A 33.1525,B 20.255,C -0.8604,E1 20.4025,E2 414.5951} C_DIS
LIN {X 103.6553,Y 71.4321,Z 147,A 31.7358,B 20.2549,C -0.8629,E1 20.4047,E2 415.9958} C_DIS
LIN {X 105.3731,Y 68.8736,Z 147,A 30.2692,B 20.2551,C -0.8567,E1 20.407,E2 417.4711} C_DIS
LIN {X 107.1846,Y 66.0183,Z 147,A 28.8152,B 20.2551,C -0.8562,E1 20.4091,E2 418.9171} C_DIS
LIN {X 108.62,Y 63.6287,Z 147,A 27.5053,B 20.2553,C -0.8512,E1 20.411,E2 420.2328} C_DIS
LIN {X 110.2839,Y 60.6999,Z 147,A 25.8628,B 20.2557,C -0.8426,E1 20.4133,E2 421.8894} C_DIS
LIN {X 112.11,Y 57.2519,Z 147,A 24.175,B 20.2557,C -0.8414,E1 20.4154,E2 423.5692} C_DIS
LIN {X 113.6837,Y 54.06,Z 147,A 22.6515,B 20.2557,C -0.841,E1 20.4173,E2 425.0836} C_DIS
LIN {X 114.9742,Y 51.258,Z 147,A 21.2586,B 20.2559,C -0.8375,E1 20.4189,E2 426.4769} C_DIS
LIN {X 116.2025,Y 48.4089,Z 147,A 19.8581,B 20.256,C -0.834,E1 20.4204,E2 427.8778} C_DIS
LIN {X 117.4474,Y 45.3062,Z 147,A 18.3465,B 20.2562,C -0.8301,E1 20.4219,E2 429.3901} C_DIS
LIN {X 118.5199,Y 42.4212,Z 147,A 16.9546,B 20.2563,C -0.8264,E1 20.4233,E2 430.7828} C_DIS
LIN {X 119.414,Y 39.834,Z 147,A 15.6986,B 20.2565,C -0.8223,E1 20.4244,E2 432.0415} C_DIS
LIN {X 120.4636,Y 36.5387,Z 147,A 14.1593,B 20.2566,C -0.8192,E1 20.4257,E2 433.5789} C_DIS
LIN {X 121.2512,Y 33.8322,Z 147,A 12.8859,B 20.2567,C -0.8157,E1 20.4267,E2 434.8529} C_DIS
LIN {X 122.0441,Y 30.85,Z 147,A 11.4974,B 20.2569,C -0.8122,E1 20.4276,E2 436.2414} C_DIS
LIN {X 122.8246,Y 27.583,Z 147,A 9.979,B 20.257,C -0.808,E1 20.4286,E2 437.7608} C_DIS
LIN {X 123.4335,Y 24.7149,Z 147,A 8.6661,B 20.2572,C -0.8049,E1 20.4293,E2 439.0731} C_DIS
LIN {X 124.0312,Y 21.5221,Z 147,A 7.2015,B 20.2573,C -0.8009,E1 20.4301,E2 440.5382} C_DIS
LIN {X 124.4762,Y 18.7728,Z 147,A 5.8745,B 20.2575,C -0.7945,E1 20.4306,E2 441.8738} C_DIS
LIN {X 124.9051,Y 15.675,Z 147,A 4.5134,B 20.2576,C -0.7927,E1 20.4311,E2 443.2299} C_DIS
LIN {X 125.2781,Y 12.3294,Z 147,A 2.8987,B 20.2579,C -0.7845,E1 20.4316,E2 444.8561} C_DIS
LIN {X 125.6064,Y 8.3639,Z 147,A 1.1541,B 20.258,C -0.7816,E1 20.432,E2 446.5959} C_DIS
LIN {X 125.7886,Y 4.8769,Z 147,A -0.4125,B 20.2582,C -0.7776,E1 20.4322,E2 448.1622} C_DIS
LIN {X 125.8707,Y 1.7949,Z 147,A -1.7246,B 20.2582,C -0.7771,E1 20.4322,E2 449.466} C_DIS
LIN {X 125.8747,Y -1.5513,Z 147,A -3.2689,B 20.2584,C -0.7714,E1 20.4322,E2 451.0151} C_DIS
LIN {X 125.8086,Y -4.3638,Z 147,A -4.6375,B 20.2587,C -0.7636,E1 20.4322,E2 452.3958} C_DIS
LIN {X 125.6633,Y -7.4408,Z 147,A -5.9555,B 20.2587,C -0.7627,E1 20.4319,E2 453.7063} C_DIS
LIN {X 125.419,Y -10.8001,Z 147,A -7.4162,B 20.2587,C -0.761,E1 20.4316,E2 455.1611} C_DIS
LIN {X 125.0869,Y -14.1517,Z 147,A -9.1327,B 20.2592,C -0.7483,E1 20.4311,E2 456.901} C_DIS
LIN {X 124.5604,Y -18.2036,Z 147,A -10.8409,B 20.2592,C -0.7489,E1 20.4304,E2 458.5948} C_DIS
LIN {X 124.0931,Y -21.1568,Z 147,A -12.1796,B 20.2593,C -0.7456,E1 20.4298,E2 459.9331} C_DIS
LIN {X 123.4641,Y -24.5645,Z 147,A -13.6526,B 20.2593,C -0.7451,E1 20.4291,E2 461.3966} C_DIS
LIN {X 122.8846,Y -27.3204,Z 147,A -14.9982,B 20.2596,C -0.7384,E1 20.4283,E2 462.7516} C_DIS
LIN {X 122.1772,Y -30.3256,Z 147,A -16.498,B 20.2599,C -0.73,E1 20.4273,E2 464.2645} C_DIS
LIN {X 121.3245,Y -33.57,Z 147,A -17.9254,B 20.2599,C -0.7296,E1 20.4263,E2 465.683} C_DIS
LIN {X 120.5451,Y -36.2725,Z 147,A -19.1952,B 20.26,C -0.7261,E1 20.4253,E2 466.9536} C_DIS
LIN {X 119.3638,Y -39.9848,Z 147,A -20.9996,B 20.2602,C -0.7193,E1 20.4237,E2 468.7644} C_DIS
LIN {X 118.0841,Y -43.6223,Z 147,A -22.6923,B 20.2603,C -0.7167,E1 20.4221,E2 470.4528} C_DIS
LIN {X 116.9805,Y -46.5012,Z 147,A -24.2307,B 20.2607,C -0.7067,E1 20.4205,E2 472.0089} C_DIS
LIN {X 115.3301,Y -50.4549,Z 147,A -26.1544,B 20.2608,C -0.7021,E1 20.4184,E2 473.9326} C_DIS
LIN {X 113.8,Y -53.8166,Z 147,A -27.6854,B 20.2608,C -0.7035,E1 20.4166,E2 475.4492} C_DIS
LIN {X 112.4479,Y -56.5881,Z 147,A -29.0761,B 20.2608,C -0.7,E1 20.4149,E2 476.8406} C_DIS
LIN {X 111.1563,Y -59.0855,Z 147,A -30.3037,B 20.2609,C -0.6985,E1 20.4133,E2 478.0643} C_DIS
LIN {X 109.5232,Y -62.062,Z 147,A -31.8522,B 20.2611,C -0.694,E1 20.4112,E2 479.6156} C_DIS
LIN {X 108.1086,Y -64.4937,Z 147,A -33.1594,B 20.2612,C -0.6892,E1 20.4094,E2 480.9278} C_DIS
LIN {X 106.4989,Y -67.1186,Z 147,A -34.4742,B 20.2612,C -0.689,E1 20.4074,E2 482.2349} C_DIS
LIN {X 104.6676,Y -69.9399,Z 147,A -36.0711,B 20.2615,C -0.682,E1 20.405,E2 483.8418} C_DIS
LIN {X 102.9233,Y -72.4825,Z 147,A -37.39,B 20.2615,C -0.6818,E1 20.4029,E2 485.153} C_DIS
LIN {X 101.116,Y -74.9835,Z 147,A -38.8544,B 20.2617,C -0.6756,E1 20.4005,E2 486.6265} C_DIS
LIN {X 98.7575,Y -78.0641,Z 147,A -40.6424,B 20.2619,C -0.6701,E1 20.3974,E2 488.4197} C_DIS
LIN {X 96.3219,Y -81.0495,Z 147,A -42.4874,B 20.2621,C -0.6618,E1 20.3941,E2 490.2778} C_DIS
LIN {X 93.3701,Y -84.4332,Z 147,A -44.424,B 20.2621,C -0.6612,E1 20.3905,E2 492.2051} C_DIS
LIN {X 90.6269,Y -87.3713,Z 147,A -46.353,B 20.2624,C -0.6526,E1 20.3868,E2 494.1482} C_DIS
LIN {X 87.8169,Y -90.1955,Z 147,A -48.1443,B 20.2625,C -0.6493,E1 20.3832,E2 495.9395} C_DIS
LIN {X 84.5628,Y -93.2525,Z 147,A -50.1658,B 20.2626,C -0.6451,E1 20.3791,E2 497.9627} C_DIS
LIN {X 81.1409,Y -96.2452,Z 147,A -52.1148,B 20.2626,C -0.6455,E1 20.375,E2 499.9007} C_DIS
LIN {X 78.0542,Y -98.7653,Z 147,A -54.0281,B 20.2629,C -0.6376,E1 20.3708,E2 501.8279} C_DIS
LIN {X 74.9956,Y -101.1069,Z 147,A -55.5841,B 20.2627,C -0.6422,E1 20.3673,E2 503.3636} C_DIS
LIN {X 72.4983,Y -102.9121,Z 147,A -56.9713,B 20.2627,C -0.64,E1 20.3642,E2 504.7508} C_DIS
LIN {X 70.1545,Y -104.5244,Z 147,A -58.3098,B 20.2629,C -0.6357,E1 20.3611,E2 506.096} C_DIS
LIN {X 67.3475,Y -106.3544,Z 147,A -59.8306,B 20.2629,C -0.633,E1 20.3575,E2 507.6181} C_DIS
LIN {X 64.4689,Y -108.1234,Z 147,A -61.4903,B 20.2632,C -0.6253,E1 20.3535,E2 509.2937} C_DIS
LIN {X 60.9373,Y -110.1524,Z 147,A -63.2096,B 20.2632,C -0.6276,E1 20.3494,E2 510.9997} C_DIS
LIN {X 58.5719,Y -111.426,Z 147,A -64.502,B 20.2633,C -0.6228,E1 20.3462,E2 512.3015} C_DIS
LIN {X 55.6373,Y -112.9199,Z 147,A -65.9076,B 20.2633,C -0.6242,E1 20.3427,E2 513.6981} C_DIS
LIN {X 52.6458,Y -114.3455,Z 147,A -67.409,B 20.2633,C -0.6222,E1 20.3389,E2 515.2004} C_DIS
LIN {X 49.8296,Y -115.6004,Z 147,A -68.8219,B 20.2633,C -0.6198,E1 20.3353,E2 516.6158} C_DIS
LIN {X 46.9853,Y -116.7854,Z 147,A -70.2614,B 20.2635,C -0.6164,E1 20.3315,E2 518.0611} C_DIS
LIN {X 43.8615,Y -117.9945,Z 147,A -71.7391,B 20.2635,C -0.6163,E1 20.3277,E2 519.5349} C_DIS
LIN {X 40.9587,Y -119.0333,Z 147,A -73.0954,B 20.2635,C -0.6165,E1 20.3241,E2 520.8873} C_DIS
LIN {X 38.2895,Y -119.9182,Z 147,A -74.4612,B 20.2636,C -0.6115,E1 20.3205,E2 522.2641} C_DIS
LIN {X 35.0619,Y -120.9017,Z 147,A -76.0123,B 20.2636,C -0.6092,E1 20.3163,E2 523.8183} C_DIS
LIN {X 30.8344,Y -122.0481,Z 147,A -77.9685,B 20.2637,C -0.6088,E1 20.311,E2 525.7721} C_DIS
LIN {X 27.5747,Y -122.8264,Z 147,A -79.4497,B 20.2637,C -0.6092,E1 20.307,E2 527.2495} C_DIS
LIN {X 24.5565,Y -123.4657,Z 147,A -80.8326,B 20.2637,C -0.6089,E1 20.3032,E2 528.631} C_DIS
LIN {X 21.524,Y -124.0309,Z 147,A -82.2406,B 20.2637,C -0.6076,E1 20.2993,E2 530.0406} C_DIS
LIN {X 18.7065,Y -124.4865,Z 147,A -83.6053,B 20.2638,C -0.6041,E1 20.2956,E2 531.4138} C_DIS
LIN {X 15.6577,Y -124.9074,Z 147,A -84.9454,B 20.2638,C -0.6057,E1 20.2919,E2 532.7479} C_DIS
LIN {X 12.3357,Y -125.2775,Z 147,A -86.4788,B 20.2638,C -0.6045,E1 20.2876,E2 534.2836} C_DIS
LIN {X 9.5335,Y -125.5221,Z 147,A -87.8242,B 20.2639,C -0.6013,E1 20.2838,E2 535.6373} C_DIS
LIN {X 6.1723,Y -125.7317,Z 147,A -89.2309,B 20.2638,C -0.6057,E1 20.2799,E2 537.0304} C_DIS
LIN {X 3.0742,Y -125.8463,Z 147,A -90.6524,B 20.2638,C -0.6049,E1 20.276,E2 538.4539} C_DIS
LIN {X 0.8881,Y -125.8783,Z 147,A -91.3005,B 20.2634,C -0.6185,E1 20.2743,E2 539.0628} C_DIS
Enddeposition()
LIN {X 0.9361,Y -131.9509,Z 148,A -93.0731,B 24.9683,C -1.3003,E1 25.0003,E2 539.6326} C_DIS
Startdeposition()
$VEL.CP = VEL_PRINT
LIN {X 5.0774,Y -131.8567,Z 148,A -90.5474,B 24.9664,C -1.3387,E1 25.0076,E2 537.0162} C_DIS
LIN {X 9.3469,Y -131.6231,Z 148,A -88.7099,B 24.9664,C -1.3385,E1 25.0128,E2 535.18} C_DIS
LIN {X 13.1366,Y -131.2998,Z 148,A -86.9906,B 24.9662,C -1.343,E1 25.0176,E2 533.4511} C_DIS
LIN {X 17.1503,Y -130.835,Z 148,A -85.3305,B 24.9664,C -1.3391,E1 25.0221,E2 531.8014} C_DIS
LIN {X 20.893,Y -130.2916,Z 148,A -83.5972,B 24.9661,C -1.3451,E1 25.027,E2 530.0555} C_DIS
LIN {X 24.6585,Y -129.6297,Z 148,A -82.0263,B 24.9663,C -1.3418,E1 25.0312,E2 528.4943} C_DIS
LIN {X 27.9696,Y -128.9558,Z 148,A -80.5533,B 24.9662,C -1.3434,E1 25.0353,E2 527.0193} C_DIS
LIN {X 31.9201,Y -128.0363,Z 148,A -78.7424,B 24.966,C -1.3478,E1 25.0402,E2 525.2006} C_DIS
LIN {X 35.377,Y -127.1234,Z 148,A -77.2606,B 24.966,C -1.3458,E1 25.0442,E2 523.7261} C_DIS
LIN {X 38.4651,Y -126.2233,Z 148,A -75.8741,B 24.966,C -1.3469,E1 25.0479,E2 522.3395} C_DIS
LIN {X 41.65,Y -125.2083,Z 148,A -74.4444,B 24.966,C -1.3475,E1 25.0517,E2 520.9108} C_DIS
LIN {X 44.7009,Y -124.1518,Z 148,A -73.0655,B 24.966,C -1.3481,E1 25.0553,E2 519.5333} C_DIS
LIN {X 47.4163,Y -123.141,Z 148,A -71.7492,B 24.9657,C -1.353,E1 25.0588,E2 518.2084} C_DIS
LIN {X 50.6198,Y -121.8586,Z 148,A -70.2779,B 24.9657,C -1.3537,E1 25.0626,E2 516.7386} C_DIS
LIN {X 53.6764,Y -120.5434,Z 148,A -68.8402,B 24.9656,C -1.3556,E1 25.0663,E2 515.3} C_DIS
LIN {X 56.6399,Y -119.1797,Z 148,A -67.4014,B 24.9654,C -1.3591,E1 25.0699,E2 513.8568} C_DIS
LIN {X 59.6571,Y -117.6983,Z 148,A -65.9723,B 24.9654,C -1.3599,E1 25.0735,E2 512.4295} C_DIS
LIN {X 62.9067,Y -115.9965,Z 148,A -64.2599,B 24.9649,C -1.3691,E1 25.0777,E2 510.7002} C_DIS
LIN {X 66.9225,Y -113.7265,Z 148,A -62.3045,B 24.9649,C -1.3703,E1 25.0824,E2 508.748} C_DIS
LIN {X 70.7786,Y -111.3683,Z 148,A -60.2998,B 24.9645,C -1.3764,E1 25.0872,E2 506.7353} C_DIS
LIN {X 74.4539,Y -108.945,Z 148,A -58.4311,B 24.9645,C -1.3779,E1 25.0915,E2 504.8691} C_DIS
LIN {X 77.9253,Y -106.4896,Z 148,A -56.5827,B 24.9642,C -1.382,E1 25.0957,E2 503.0177} C_DIS
LIN {X 81.4314,Y -103.8328,Z 148,A -54.6976,B 24.9641,C -1.3848,E1 25.0999,E2 501.1328} C_DIS
LIN {X 84.8338,Y -101.072,Z 148,A -52.8116,B 24.9639,C -1.3882,E1 25.104,E2 499.2459} C_DIS
LIN {X 88.2711,Y -98.0848,Z 148,A -50.8197,B 24.9636,C -1.3937,E1 25.1081,E2 497.2491} C_DIS
LIN {X 91.4485,Y -95.1296,Z 148,A -48.9346,B 24.9634,C -1.3984,E1 25.112,E2 495.3608} C_DIS
LIN {X 94.5716,Y -92.0252,Z 148,A -47.0486,B 24.9632,C -1.4017,E1 25.1157,E2 493.4748} C_DIS
LIN {X 97.5725,Y -88.8369,Z 148,A -45.1591,B 24.963,C -1.406,E1 25.1193,E2 491.5835} C_DIS
LIN {X 100.473,Y -85.5425,Z 148,A -43.4491,B 24.9633,C -1.4003,E1 25.1223,E2 489.8947} C_DIS
LIN {X 103.0231,Y -82.4541,Z 148,A -41.4473,B 24.9623,C -1.4195,E1 25.1259,E2 487.857} C_DIS
LIN {X 106.0278,Y -78.5528,Z 148,A -39.4256,B 24.9623,C -1.419,E1 25.1293,E2 485.8461} C_DIS
LIN {X 108.5495,Y -75.03,Z 148,A -37.7428,B 24.9626,C -1.4134,E1 25.132,E2 484.1847} C_DIS
LIN {X 110.3797,Y -72.3101,Z 148,A -36.1601,B 24.9619,C -1.4262,E1 25.1345,E2 482.5795} C_DIS
LIN {X 112.6697,Y -68.6877,Z 148,A -34.2521,B 24.9615,C -1.4343,E1 25.1373,E2 480.6623} C_DIS
LIN {X 114.8907,Y -64.904,Z 148,A -32.3815,B 24.9613,C -1.4381,E1 25.1399,E2 478.7924} C_DIS
LIN {X 116.9081,Y -61.191,Z 148,A -30.6666,B 24.9613,C -1.437,E1 25.1421,E2 477.089} C_DIS
LIN {X 118.4123,Y -58.2269,Z 148,A -29.2545,B 24.9612,C -1.4397,E1 25.1439,E2 475.6781} C_DIS
LIN {X 119.7726,Y -55.3746,Z 148,A -27.8776,B 24.9609,C -1.4442,E1 25.1455,E2 474.2981} C_DIS
LIN {X 121.0591,Y -52.5027,Z 148,A -26.5167,B 24.9607,C -1.4482,E1 25.1471,E2 472.9352} C_DIS
LIN {X 122.2729,Y -49.6112,Z 148,A -25.1439,B 24.9604,C -1.4531,E1 25.1485,E2 471.5584} C_DIS
LIN {X 123.5023,Y -46.4656,Z 148,A -23.6853,B 24.9602,C -1.4573,E1 25.15,E2 470.0981} C_DIS
LIN {X 124.65,Y -43.2924,Z 148,A -22.2625,B 24.9601,C -1.4596,E1 25.1513,E2 468.6778} C_DIS
LIN {X 126.6076,Y -37.1806,Z 148,A -19.4368,B 24.9595,C -1.4707,E1 25.1537,E2 465.8419} C_DIS
LIN {X 127.6546,Y -33.4146,Z 148,A -17.6672,B 24.959,C -1.4802,E1 25.155,E2 464.0601} C_DIS
LIN {X 128.4543,Y -30.198,Z 148,A -16.2221,B 24.9587,C -1.4852,E1 25.1559,E2 462.6115} C_DIS
LIN {X 129.2861,Y -26.4007,Z 148,A -14.6813,B 24.9588,C -1.4826,E1 25.1568,E2 461.0858} C_DIS
LIN {X 129.9892,Y -22.694,Z 148,A -12.937,B 24.9582,C -1.4939,E1 25.1577,E2 459.3252} C_DIS
LIN {X 130.6074,Y -18.8054,Z 148,A -11.3527,B 24.9582,C -1.4926,E1 25.1583,E2 457.7533} C_DIS
LIN {X 131.0641,Y -15.3043,Z 148,A -9.7195,B 24.9577,C -1.5032,E1 25.1589,E2 456.1047} C_DIS
LIN {X 131.4799,Y -11.179,Z 148,A -8.0197,B 24.9577,C -1.5036,E1 25.1593,E2 454.4141} C_DIS
LIN {X 131.7643,Y -7.0961,Z 148,A -6.2578,B 24.9574,C -1.5086,E1 25.1596,E2 452.6508} C_DIS
LIN {X 131.9068,Y -3.5446,Z 148,A -4.7008,B 24.957,C -1.5145,E1 25.1598,E2 451.0892} C_DIS
LIN {X 131.9558,Y 0.3789,Z 148,A -2.9335,B 24.9565,C -1.5237,E1 25.1598,E2 449.3108} C_DIS
LIN {X 131.87,Y 4.7366,Z 148,A -1.1286,B 24.9565,C -1.5251,E1 25.1596,E2 447.5134} C_DIS
LIN {X 131.6904,Y 8.3456,Z 148,A 0.4204,B 24.9562,C -1.5291,E1 25.1594,E2 445.964} C_DIS
LIN {X 131.3598,Y 12.5123,Z 148,A 2.1756,B 24.956,C -1.5318,E1 25.159,E2 444.213} C_DIS
LIN {X 130.9921,Y 15.9083,Z 148,A 3.7263,B 24.9555,C -1.5403,E1 25.1585,E2 442.6513} C_DIS
LIN {X 130.4171,Y 20.0823,Z 148,A 5.4939,B 24.9555,C -1.5428,E1 25.1578,E2 440.8882} C_DIS
LIN {X 129.7612,Y 23.9682,Z 148,A 7.2679,B 24.9549,C -1.5518,E1 25.1569,E2 439.1035} C_DIS
LIN {X 129.0082,Y 27.7271,Z 148,A 8.8222,B 24.9549,C -1.551,E1 25.156,E2 437.56} C_DIS
LIN {X 128.2481,Y 31.0534,Z 148,A 10.3466,B 24.9545,C -1.5581,E1 25.155,E2 436.0278} C_DIS
LIN {X 127.154,Y 35.2676,Z 148,A 12.1778,B 24.9544,C -1.5607,E1 25.1537,E2 434.2009} C_DIS
LIN {X 126.2171,Y 38.4855,Z 148,A 13.5962,B 24.9542,C -1.5632,E1 25.1526,E2 432.7847} C_DIS
LIN {X 125.2278,Y 41.5916,Z 148,A 15.018,B 24.9539,C -1.5679,E1 25.1513,E2 431.3599} C_DIS
LIN {X 124.1406,Y 44.7319,Z 148,A 16.43,B 24.9538,C -1.5706,E1 25.15,E2 429.9494} C_DIS
LIN {X 123.0418,Y 47.6715,Z 148,A 17.857,B 24.9533,C -1.5783,E1 25.1486,E2 428.5123} C_DIS
LIN {X 121.645,Y 51.1313,Z 148,A 19.4758,B 24.953,C -1.583,E1 25.1469,E2 426.8913} C_DIS
LIN {X 119.8903,Y 55.1201,Z 148,A 21.2969,B 24.953,C -1.5847,E1 25.1448,E2 425.0762} C_DIS
LIN {X 118.5168,Y 58.0151,Z 148,A 22.6982,B 24.9527,C -1.5892,E1 25.1431,E2 423.6717} C_DIS
LIN {X 116.9243,Y 61.16,Z 148,A 24.2099,B 24.9525,C -1.5925,E1 25.1412,E2 422.1602} C_DIS
LIN {X 114.8457,Y 64.9841,Z 148,A 26.2145,B 24.9518,C -1.6041,E1 25.1384,E2 420.1389} C_DIS
LIN {X 112.6294,Y 68.7534,Z 148,A 28.0751,B 24.9516,C -1.6072,E1 25.1358,E2 418.2805} C_DIS
LIN {X 110.3689,Y 72.3264,Z 148,A 29.925,B 24.9513,C -1.6128,E1 25.1329,E2 416.4265} C_DIS
LIN {X 107.813,Y 76.0834,Z 148,A 31.8302,B 24.9512,C -1.6142,E1 25.1299,E2 414.5273} C_DIS
LIN {X 105.0044,Y 79.9156,Z 148,A 34.4366,B 24.949,C -1.6491,E1 25.1254,E2 411.8511} C_DIS
LIN {X 101.9506,Y 83.7766,Z 148,A 36.1033,B 24.9503,C -1.6286,E1 25.1226,E2 410.2405} C_DIS
LIN {X 98.9611,Y 87.2871,Z 148,A 38.0247,B 24.9503,C -1.629,E1 25.1191,E2 408.327} C_DIS
LIN {X 95.9755,Y 90.5595,Z 148,A 39.9193,B 24.9501,C -1.6318,E1 25.1155,E2 406.434} C_DIS
LIN {X 92.8471,Y 93.7645,Z 148,A 41.8742,B 24.9498,C -1.6366,E1 25.1116,E2 404.476} C_DIS
LIN {X 89.6248,Y 96.8499,Z 148,A 43.8239,B 24.9495,C -1.6414,E1 25.1077,E2 402.523} C_DIS
LIN {X 86.3491,Y 99.781,Z 148,A 45.7317,B 24.9493,C -1.6452,E1 25.1037,E2 400.6137} C_DIS
LIN {X 82.8918,Y 102.6707,Z 148,A 47.6339,B 24.9493,C -1.6461,E1 25.0996,E2 398.7167} C_DIS
LIN {X 79.4309,Y 105.371,Z 148,A 49.3141,B 24.9498,C -1.6376,E1 25.0959,E2 397.0628} C_DIS
LIN {X 74.2632,Y 109.0754,Z 148,A 52.3476,B 24.9486,C -1.6569,E1 25.0889,E2 393.9942} C_DIS
LIN {X 70.4215,Y 111.5936,Z 148,A 54.2797,B 24.9486,C -1.6568,E1 25.0844,E2 392.0687} C_DIS
LIN {X 66.6459,Y 113.889,Z 148,A 56.2052,B 24.9484,C -1.66,E1 25.0798,E2 390.1413} C_DIS
LIN {X 62.9338,Y 115.9817,Z 148,A 58.4467,B 24.9469,C -1.6835,E1 25.0742,E2 387.851} C_DIS
LIN {X 59.1931,Y 117.9346,Z 148,A 59.8715,B 24.9481,C -1.6642,E1 25.0707,E2 386.4756} C_DIS
LIN {X 55.732,Y 119.6073,Z 148,A 61.4112,B 24.9484,C -1.6595,E1 25.0669,E2 384.9511} C_DIS
LIN {X 52.7016,Y 120.9732,Z 148,A 62.9176,B 24.9481,C -1.6645,E1 25.063,E2 383.4366} C_DIS
LIN {X 49.4735,Y 122.3284,Z 148,A 64.3841,B 24.9481,C -1.6633,E1 25.0592,E2 381.9763} C_DIS
LIN {X 46.4529,Y 123.5071,Z 148,A 65.7861,B 24.9481,C -1.6644,E1 25.0556,E2 380.5747} C_DIS
LIN {X 43.2987,Y 124.6478,Z 148,A 67.2264,B 24.9481,C -1.6649,E1 25.0518,E2 379.1362} C_DIS
LIN {X 40.3239,Y 125.6418,Z 148,A 68.6337,B 24.9478,C -1.6684,E1 25.0481,E2 377.7233} C_DIS
LIN {X 37.1745,Y 126.6094,Z 148,A 70.0358,B 24.9478,C -1.668,E1 25.0443,E2 376.3245} C_DIS
LIN {X 31.5834,Y 128.1204,Z 148,A 72.6458,B 24.9475,C -1.6745,E1 25.0372,E2 373.7031} C_DIS
LIN {X 27.8566,Y 128.9802,Z 148,A 74.2218,B 24.9477,C -1.671,E1 25.033,E2 372.1376} C_DIS
LIN {X 24.9552,Y 129.573,Z 148,A 75.6029,B 24.9473,C -1.6765,E1 25.0292,E2 370.7451} C_DIS
LIN {X 20.5768,Y 130.3406,Z 148,A 77.474,B 24.9475,C -1.6741,E1 25.024,E2 368.8816} C_DIS
LIN {X 16.97,Y 130.8586,Z 148,A 79.0771,B 24.9474,C -1.6756,E1 25.0196,E2 367.2762} C_DIS
LIN {X 12.7985,Y 131.3323,Z 148,A 80.8525,B 24.9475,C -1.6734,E1 25.0147,E2 365.5072} C_DIS
LIN {X 9.3809,Y 131.6206,Z 148,A 82.4087,B 24.9473,C -1.677,E1 25.0103,E2 363.9434} C_DIS
LIN {X 5.3807,Y 131.8448,Z 148,A 84.0906,B 24.9475,C -1.6739,E1 25.0056,E2 362.2692} C_DIS
LIN {X 1.4994,Y 131.9477,Z 148,A 85.8613,B 24.9472,C -1.678,E1 25.0007,E2 360.4891} C_DIS
LIN {X -2.443,Y 131.932,Z 148,A 87.5594,B 24.9473,C -1.6769,E1 24.9959,E2 358.7935} C_DIS
LIN {X -6.5359,Y 131.7924,Z 148,A 89.2397,B 24.9477,C -1.6714,E1 24.9913,E2 357.1261} C_DIS
LIN {X -10.333,Y 131.5511,Z 148,A 91.0439,B 24.9472,C -1.6784,E1 24.9862,E2 355.3046} C_DIS
LIN {X -14.2437,Y 131.1833,Z 148,A 92.5921,B 24.9478,C -1.6695,E1 24.982,E2 353.7766} C_DIS
LIN {X -20.1891,Y 130.4006,Z 148,A 95.0896,B 24.9482,C -1.6624,E1 24.9751,E2 351.2939} C_DIS
LIN {X -26.0842,Y 129.3505,Z 148,A 97.6195,B 24.9486,C -1.6568,E1 24.9682,E2 348.7747} C_DIS
LIN {X -29.1993,Y 128.683,Z 148,A 99.1863,B 24.9481,C -1.6648,E1 24.9639,E2 347.1871} C_DIS
LIN {X -32.3953,Y 127.9157,Z 148,A 100.6334,B 24.9481,C -1.6644,E1 24.9599,E2 345.7388} C_DIS
LIN {X -35.5934,Y 127.0629,Z 148,A 102.1022,B 24.9481,C -1.6644,E1 24.956,E2 344.2676} C_DIS
LIN {X -39.5766,Y 125.8806,Z 148,A 103.9281,B 24.9481,C -1.6634,E1 24.9511,E2 342.441} C_DIS
LIN {X -42.9489,Y 124.7691,Z 148,A 105.4099,B 24.9485,C -1.6585,E1 24.9472,E2 340.968} C_DIS
LIN {X -46.1762,Y 123.6107,Z 148,A 106.8991,B 24.9485,C -1.6566,E1 24.9433,E2 339.4805} C_DIS
LIN {X -49.2427,Y 122.4214,Z 148,A 108.3176,B 24.9487,C -1.6541,E1 24.9396,E2 338.0647} C_DIS
LIN {X -52.0993,Y 121.2336,Z 148,A 109.7129,B 24.9487,C -1.6547,E1 24.936,E2 336.6647} C_DIS
LIN {X -55.1785,Y 119.8633,Z 148,A 111.1973,B 24.9487,C -1.6535,E1 24.9322,E2 335.1797} C_DIS
LIN {X -58.2496,Y 118.4011,Z 148,A 112.6485,B 24.949,C -1.6499,E1 24.9286,E2 333.7334} C_DIS
LIN {X -60.9579,Y 117.0305,Z 148,A 114.007,B 24.949,C -1.6496,E1 24.9252,E2 332.3717} C_DIS
LIN {X -64.7334,Y 114.9866,Z 148,A 115.9339,B 24.949,C -1.6494,E1 24.9205,E2 330.4398} C_DIS
LIN {X -68.4933,Y 112.7876,Z 148,A 117.8491,B 24.9492,C -1.6471,E1 24.9159,E2 328.5243} C_DIS
LIN {X -72.2607,Y 110.4122,Z 148,A 119.5521,B 24.9501,C -1.632,E1 24.912,E2 326.8518} C_DIS
LIN {X -75.864,Y 107.9678,Z 148,A 121.7056,B 24.9495,C -1.641,E1 24.9069,E2 324.6694} C_DIS
LIN {X -79.5192,Y 105.3044,Z 148,A 123.6505,B 24.9499,C -1.6359,E1 24.9026,E2 322.7297} C_DIS
LIN {X -83.0435,Y 102.5484,Z 148,A 125.6215,B 24.95,C -1.633,E1 24.8983,E2 320.7583} C_DIS
LIN {X -86.4333,Y 99.7085,Z 148,A 127.5358,B 24.9503,C -1.6283,E1 24.8942,E2 318.8478} C_DIS
LIN {X -89.6346,Y 96.8407,Z 148,A 129.4148,B 24.9505,C -1.6245,E1 24.8903,E2 316.9703} C_DIS
LIN {X -92.7064,Y 93.9043,Z 148,A 131.8001,B 24.9492,C -1.6465,E1 24.8855,E2 314.5225} C_DIS
LIN {X -96.117,Y 90.4095,Z 148,A 133.2441,B 24.9515,C -1.6081,E1 24.8829,E2 313.1639} C_DIS
LIN {X -99.1531,Y 87.0698,Z 148,A 135.4102,B 24.9512,C -1.613,E1 24.8788,E2 310.9764} C_DIS
LIN {X -102.0092,Y 83.7049,Z 148,A 137.3088,B 24.9516,C -1.607,E1 24.8754,E2 309.0832} C_DIS
LIN {X -104.7726,Y 80.2186,Z 148,A 139.2404,B 24.9519,C -1.6018,E1 24.8721,E2 307.155} C_DIS
LIN {X -107.4995,Y 76.5262,Z 148,A 141.243,B 24.9522,C -1.5967,E1 24.8688,E2 305.1548} C_DIS
LIN {X -109.2947,Y 73.9391,Z 148,A 142.7417,B 24.9521,C -1.5992,E1 24.8664,E2 303.6428} C_DIS
LIN {X -112.0558,Y 69.6837,Z 148,A 144.8178,B 24.9528,C -1.5867,E1 24.8634,E2 301.5859} C_DIS
LIN {X -114.3382,Y 65.8724,Z 148,A 146.7909,B 24.953,C -1.5831,E1 24.8606,E2 299.6111} C_DIS
LIN {X -116.4042,Y 62.1491,Z 148,A 148.6828,B 24.9532,C -1.5797,E1 24.858,E2 297.7174} C_DIS
LIN {X -118.2049,Y 58.6473,Z 148,A 150.3003,B 24.9538,C -1.57,E1 24.856,E2 296.1141} C_DIS
LIN {X -119.7001,Y 55.5313,Z 148,A 151.7603,B 24.9542,C -1.5635,E1 24.8543,E2 294.6618} C_DIS
LIN {X -121.0666,Y 52.4855,Z 148,A 153.2172,B 24.9544,C -1.5593,E1 24.8527,E2 293.2067} C_DIS
LIN {X -122.3093,Y 49.5209,Z 148,A 154.6273,B 24.9547,C -1.5557,E1 24.8512,E2 291.7975} C_DIS
LIN {X -123.537,Y 46.3731,Z 148,A 156.0792,B 24.955,C -1.5503,E1 24.8497,E2 290.3502} C_DIS
LIN {X -124.65,Y 43.2924,Z 148,A 157.5219,B 24.9552,C -1.5468,E1 24.8484,E2 288.9078} C_DIS
LIN {X -125.6454,Y 40.3128,Z 148,A 158.9227,B 24.9553,C -1.5442,E1 24.8472,E2 287.5051} C_DIS
LIN {X -126.6494,Y 37.0378,Z 148,A 160.4263,B 24.9556,C -1.5402,E1 24.846,E2 286.0025} C_DIS
LIN {X -127.6814,Y 33.3141,Z 148,A 162.2319,B 24.9556,C -1.5408,E1 24.8446,E2 284.1848} C_DIS
LIN {X -128.4786,Y 30.0942,Z 148,A 164.1552,B 24.9544,C -1.5595,E1 24.8434,E2 282.2057} C_DIS
LIN {X -129.4762,Y 25.4615,Z 148,A 165.5742,B 24.9566,C -1.5219,E1 24.8427,E2 280.8679} C_DIS
LIN {X -130.5871,Y 18.9473,Z 148,A 168.9033,B 24.9559,C -1.5346,E1 24.8412,E2 277.4888} C_DIS
LIN {X -131.0618,Y 15.324,Z 148,A 170.1629,B 24.9571,C -1.5136,E1 24.8407,E2 276.2717} C_DIS
LIN {X -131.4409,Y 11.6417,Z 148,A 172.0018,B 24.9567,C -1.5194,E1 24.8403,E2 274.4079} C_DIS
LIN {X -131.7826,Y 6.7305,Z 148,A 173.9243,B 24.9577,C -1.502,E1 24.8399,E2 272.5154} C_DIS
LIN {X -131.9309,Y 2.509,Z 148,A 175.7489,B 24.9581,C -1.4955,E1 24.8398,E2 270.6953} C_DIS
LIN {X -131.9333,Y -2.3645,Z 148,A 177.9352,B 24.9583,C -1.4919,E1 24.8398,E2 268.5044} C_DIS
LIN {X -131.7873,Y -6.6373,Z 148,A 179.7693,B 24.9587,C -1.4847,E1 24.8401,E2 266.6764} C_DIS
LIN {X -131.1977,Y -14.1102,Z 148,A -176.9473,B 24.9592,C -1.4754,E1 24.8409,E2 263.3955} C_DIS
LIN {X -130.6915,Y -18.217,Z 148,A -175.1127,B 24.9594,C -1.4714,E1 24.8415,E2 261.5595} C_DIS
LIN {X -130.1427,Y -21.7894,Z 148,A -173.5964,B 24.9599,C -1.4637,E1 24.8422,E2 260.0523} C_DIS
LIN {X -129.4393,Y -25.6479,Z 148,A -171.7717,B 24.9599,C -1.4641,E1 24.8431,E2 258.2159} C_DIS
LIN {X -128.6637,Y -29.2838,Z 148,A -170.2583,B 24.9604,C -1.4542,E1 24.844,E2 256.7173} C_DIS
LIN {X -127.919,Y -32.3822,Z 148,A -168.8803,B 24.9606,C -1.4495,E1 24.845,E2 255.3423} C_DIS
LIN {X -127.0821,Y -35.5249,Z 148,A -167.4436,B 24.9608,C -1.4463,E1 24.846,E2 253.905} C_DIS
LIN {X -126.1561,Y -38.6846,Z 148,A -165.9951,B 24.961,C -1.4428,E1 24.8472,E2 252.4565} C_DIS
LIN {X -125.0096,Y -42.2468,Z 148,A -164.2621,B 24.961,C -1.4431,E1 24.8487,E2 250.7129} C_DIS
LIN {X -123.6599,Y -46.0449,Z 148,A -162.6024,B 24.9615,C -1.4334,E1 24.8503,E2 249.067} C_DIS
LIN {X -122.4439,Y -49.1868,Z 148,A -161.1438,B 24.9618,C -1.4288,E1 24.8518,E2 247.6111} C_DIS
LIN {X -121.1942,Y -52.1904,Z 148,A -159.7153,B 24.9619,C -1.4254,E1 24.8533,E2 246.1827} C_DIS
LIN {X -119.8475,Y -55.2126,Z 148,A -158.2521,B 24.9621,C -1.4225,E1 24.855,E2 244.7184} C_DIS
LIN {X -118.4242,Y -58.2028,Z 148,A -156.8057,B 24.9623,C -1.4188,E1 24.8568,E2 243.2731} C_DIS
LIN {X -116.8967,Y -61.2128,Z 148,A -155.3315,B 24.9625,C -1.4151,E1 24.8587,E2 241.7998} C_DIS
LIN {X -114.8347,Y -65.0037,Z 148,A -153.3302,B 24.9625,C -1.416,E1 24.8614,E2 239.7857} C_DIS
LIN {X -112.6527,Y -68.7155,Z 148,A -151.4516,B 24.9627,C -1.4114,E1 24.8641,E2 237.9084} C_DIS
LIN {X -110.2835,Y -72.4562,Z 148,A -149.5664,B 24.963,C -1.4045,E1 24.8669,E2 236.0302} C_DIS
LIN {X -107.8366,Y -76.05,Z 148,A -147.687,B 24.9633,C -1.3992,E1 24.8699,E2 234.1542} C_DIS
LIN {X -105.2933,Y -79.534,Z 148,A -145.7944,B 24.9635,C -1.3954,E1 24.8731,E2 232.2614} C_DIS
LIN {X -102.5649,Y -83.023,Z 148,A -143.8292,B 24.9637,C -1.3928,E1 24.8765,E2 230.2932} C_DIS
LIN {X -99.945,Y -86.1587,Z 148,A -142.0436,B 24.9639,C -1.3892,E1 24.8797,E2 228.5081} C_DIS
LIN {X -96.9076,Y -89.562,Z 148,A -140.0865,B 24.9641,C -1.3835,E1 24.8834,E2 226.5559} C_DIS
LIN {X -93.8748,Y -92.7361,Z 148,A -138.1136,B 24.9641,C -1.3826,E1 24.8872,E2 224.5767} C_DIS
LIN {X -90.7317,Y -95.8131,Z 148,A -136.2004,B 24.9644,C -1.3787,E1 24.8911,E2 222.6648} C_DIS
LIN {X -87.3743,Y -98.884,Z 148,A -134.2658,B 24.9647,C -1.3726,E1 24.8951,E2 220.7369} C_DIS
LIN {X -83.9749,Y -101.787,Z 148,A -132.2832,B 24.9647,C -1.3709,E1 24.8993,E2 218.7508} C_DIS
LIN {X -80.5203,Y -104.5417,Z 148,A -130.3305,B 24.9649,C -1.369,E1 24.9036,E2 216.7952} C_DIS
LIN {X -76.9904,Y -107.1676,Z 148,A -128.4294,B 24.9651,C -1.3652,E1 24.9079,E2 214.8965} C_DIS
LIN {X -73.4056,Y -109.6538,Z 148,A -126.5446,B 24.9653,C -1.3616,E1 24.9123,E2 213.0141} C_DIS
LIN {X -69.649,Y -112.0774,Z 148,A -124.6098,B 24.9654,C -1.3582,E1 24.9168,E2 211.0812} C_DIS
LIN {X -65.7523,Y -114.4077,Z 148,A -121.4346,B 24.9624,C -1.4169,E1 24.9249,E2 207.7571} C_DIS
LIN {X -58.4842,Y -118.2854,Z 148,A -119.2268,B 24.9663,C -1.3421,E1 24.93,E2 205.7211} C_DIS
LIN {X -55.6243,Y -119.6572,Z 148,A -117.7387,B 24.9661,C -1.346,E1 24.9338,E2 204.2198} C_DIS
LIN {X -52.4626,Y -121.0765,Z 148,A -116.3206,B 24.9664,C -1.3399,E1 24.9373,E2 202.8128} C_DIS
LIN {X -49.5028,Y -122.3166,Z 148,A -114.8645,B 24.9663,C -1.3417,E1 24.9411,E2 201.3493} C_DIS
LIN {X -46.4581,Y -123.5052,Z 148,A -113.4383,B 24.9663,C -1.3406,E1 24.9448,E2 199.9226} C_DIS
LIN {X -43.3657,Y -124.6246,Z 148,A -112.0107,B 24.9664,C -1.3394,E1 24.9486,E2 198.4952} C_DIS
LIN {X -40.1582,Y -125.6948,Z 148,A -110.529,B 24.9664,C -1.3389,E1 24.9525,E2 197.0119} C_DIS
LIN {X -35.7606,Y -127.0162,Z 148,A -108.5955,B 24.9667,C -1.3343,E1 24.9577,E2 195.0859} C_DIS
LIN {X -32.8966,Y -127.7885,Z 148,A -107.2072,B 24.9664,C -1.3387,E1 24.9615,E2 193.6853} C_DIS
LIN {X -29.6028,Y -128.5909,Z 148,A -105.7489,B 24.9665,C -1.3372,E1 24.9654,E2 192.2285} C_DIS
Enddeposition()
END
